LIN {X -0.012,Y -226.198,Z 1158.241,A 0.000,B 0.000,C 90.000,E1 43.380} C_DIS
LIN {X -0.070,Y -217.479,Z 1158.220,A 0.000,B 0.000,C 90.000,E1 39.564} C_DIS
LIN {X -0.002,Y -209.401,Z 1158.198,A 0.000,B 0.000,C 90.000,E1 35.644} C_DIS
LIN {X 0.014,Y -202.068,Z 1158.176,A 0.000,B 0.000,C 90.000,E1 31.671} C_DIS
LIN {X 0.064,Y -196.716,Z 1158.158,A 0.000,B 0.000,C 90.000,E1 28.437} C_DIS
LIN {X -0.032,Y -190.859,Z 1158.135,A 0.000,B 0.000,C 90.000,E1 24.387} C_DIS
LIN {X -0.001,Y -185.887,Z 1158.112,A 0.000,B 0.000,C 90.000,E1 20.248} C_DIS
LIN {X -0.022,Y -181.921,Z 1158.089,A 0.000,B 0.000,C 90.000,E1 16.079} C_DIS
LIN {X -0.067,Y -178.946,Z 1158.066,A 0.000,B 0.000,C 90.000,E1 11.883} C_DIS
LIN {X 0.040,Y -176.545,Z 1158.033,A 0.000,B 0.000,C 90.000,E1 5.910} C_DIS
LIN {X -0.034,Y -177.523,Z 1157.969,A 0.000,B 0.000,C 90.000,E1 354.432} C_DIS
LIN {X -0.032,Y -180.412,Z 1157.941,A 0.000,B 0.000,C 90.000,E1 349.342} C_DIS
LIN {X 0.053,Y -183.846,Z 1157.917,A 0.000,B 0.000,C 90.000,E1 345.102} C_DIS
LIN {X 0.088,Y -188.207,Z 1157.894,A 0.000,B 0.000,C 90.000,E1 340.913} C_DIS
LIN {X 0.033,Y -193.296,Z 1157.871,A 0.000,B 0.000,C 90.000,E1 336.794} C_DIS
LIN {X -0.094,Y -199.221,Z 1157.848,A 0.000,B 0.000,C 90.000,E1 332.743} C_DIS
LIN {X 0.072,Y -205.805,Z 1157.826,A 0.000,B 0.000,C 90.000,E1 328.663} C_DIS
LIN {X 0.075,Y -213.259,Z 1157.804,A 0.000,B 0.000,C 90.000,E1 324.689} C_DIS
LIN {X -0.021,Y -220.064,Z 1157.786,A 0.000,B 0.000,C 90.000,E1 321.582} C_DIS
LIN {X 0.021,Y -227.922,Z 1157.769,A 0.000,B 0.000,C 90.000,E1 318.485} C_DIS
LIN {X 0.025,Y -237.826,Z 1157.750,A 0.000,B 0.000,C 90.000,E1 315.081} C_DIS
LIN {X -0.014,Y -247.747,Z 1157.734,A 0.000,B 0.000,C 90.000,E1 312.123} C_DIS
LIN {X 0.041,Y -257.436,Z 1157.720,A 0.000,B 0.000,C 90.000,E1 309.564} C_DIS
LIN {X -0.005,Y -267.881,Z 1157.706,A 0.000,B 0.000,C 90.000,E1 307.076} C_DIS
LIN {X 0.126,Y -282.892,Z 1157.689,A 0.000,B 0.000,C 90.000,E1 303.913} C_DIS
LIN {X 0.086,Y -299.824,Z 1157.672,A 0.000,B 0.000,C 90.000,E1 300.875} C_DIS
LIN {X 0.078,Y -312.165,Z 1157.661,A 0.000,B 0.000,C 90.000,E1 298.899} C_DIS
LIN {X -0.128,Y -325.531,Z 1157.650,A 0.000,B 0.000,C 90.000,E1 297.001} C_DIS
LIN {X 0.004,Y -337.614,Z 1157.641,A 0.000,B 0.000,C 90.000,E1 295.412} C_DIS
LIN {X 0.021,Y -353.190,Z 1157.631,A 0.000,B 0.000,C 90.000,E1 293.567} C_DIS
LIN {X -0.118,Y -368.772,Z 1157.622,A 0.000,B 0.000,C 90.000,E1 291.972} C_DIS
LIN {X 0.035,Y -387.878,Z 1157.612,A 0.000,B 0.000,C 90.000,E1 290.174} C_DIS
LIN {X -0.171,Y -398.718,Z 1157.607,A 0.000,B 0.000,C 90.000,E1 289.214} C_DIS
LIN {X 0.062,Y -409.265,Z 1157.601,A 0.000,B 0.000,C 90.000,E1 288.181} C_DIS
LIN {X -0.151,Y -416.945,Z 1157.597,A 0.000,B 0.000,C 90.000,E1 287.457} C_DIS
LIN {X 0.059,Y -426.961,Z 1157.591,A 0.000,B 0.000,C 90.000,E1 286.386} C_DIS
LIN {X -0.111,Y -434.256,Z 1157.587,A 0.000,B 0.000,C 90.000,E1 285.607} C_DIS
LIN {X 0.144,Y -440.949,Z 1157.582,A 0.000,B 0.000,C 90.000,E1 284.773} C_DIS
LIN {X -0.071,Y -446.923,Z 1157.578,A 0.000,B 0.000,C 90.000,E1 284.008} C_DIS
LIN {X -0.137,Y -452.227,Z 1157.573,A 0.000,B 0.000,C 90.000,E1 283.231} C_DIS
LIN {X 0.186,Y -456.836,Z 1157.569,A 0.000,B 0.000,C 90.000,E1 282.411} C_DIS
LIN {X 0.008,Y -460.800,Z 1157.565,A 0.000,B 0.000,C 90.000,E1 281.658} C_DIS
LIN {X -0.036,Y -464.268,Z 1157.561,A 0.000,B 0.000,C 90.000,E1 280.894} C_DIS
LIN {X -0.142,Y -467.259,Z 1157.556,A 0.000,B 0.000,C 90.000,E1 280.141} C_DIS
LIN {X 0.005,Y -468.995,Z 1157.553,A 0.000,B 0.000,C 90.000,E1 279.613} C_DIS
LIN {X 0.087,Y -470.532,Z 1157.551,A 0.000,B 0.000,C 90.000,E1 279.095} C_DIS
LIN {X -0.214,Y -471.856,Z 1157.548,A 0.000,B 0.000,C 90.000,E1 278.624} C_DIS
LIN {X -0.111,Y -472.903,Z 1157.545,A 0.000,B 0.000,C 90.000,E1 278.106} C_DIS
LIN {X 0.001,Y -473.652,Z 1157.542,A 0.000,B 0.000,C 90.000,E1 277.587} C_DIS
LIN {X 0.122,Y -474.004,Z 1157.539,A 0.000,B 0.000,C 90.000,E1 277.068} C_DIS
LIN {X -0.222,Y -474.027,Z 1157.536,A 0.000,B 0.000,C 90.000,E1 276.606} C_DIS
LIN {X -0.095,Y -473.593,Z 1157.534,A 0.000,B 0.000,C 90.000,E1 276.087} C_DIS
LIN {X 0.033,Y -472.728,Z 1157.531,A 0.000,B 0.000,C 90.000,E1 275.568} C_DIS
LIN {X 0.156,Y -471.403,Z 1157.528,A 0.000,B 0.000,C 90.000,E1 275.049} C_DIS
LIN {X -0.196,Y -469.630,Z 1157.525,A 0.000,B 0.000,C 90.000,E1 274.588} C_DIS
LIN {X -0.123,Y -467.288,Z 1157.523,A 0.000,B 0.000,C 90.000,E1 274.073} C_DIS
LIN {X -0.032,Y -464.287,Z 1157.520,A 0.000,B 0.000,C 90.000,E1 273.555} C_DIS
LIN {X 0.039,Y -460.432,Z 1157.517,A 0.000,B 0.000,C 90.000,E1 273.037} C_DIS
LIN {X -0.177,Y -458.255,Z 1157.516,A 0.000,B 0.000,C 90.000,E1 272.808} C_DIS
LIN {X -0.080,Y -452.850,Z 1157.513,A 0.000,B 0.000,C 90.000,E1 272.293} C_DIS
LIN {X -0.220,Y -449.791,Z 1157.511,A 0.000,B 0.000,C 90.000,E1 272.064} C_DIS
LIN {X -0.132,Y -446.731,Z 1157.510,A 0.000,B 0.000,C 90.000,E1 271.835} C_DIS
LIN {X -0.085,Y -440.020,Z 1157.508,A 0.000,B 0.000,C 90.000,E1 271.432} C_DIS
LIN {X 0.061,Y -433.083,Z 1157.506,A 0.000,B 0.000,C 90.000,E1 271.088} C_DIS
LIN {X 0.186,Y -426.162,Z 1157.505,A 0.000,B 0.000,C 90.000,E1 270.802} C_DIS
LIN {X 0.201,Y -419.177,Z 1157.503,A 0.000,B 0.000,C 90.000,E1 270.573} C_DIS
LIN {X 0.062,Y -411.911,Z 1157.502,A 0.000,B 0.000,C 90.000,E1 270.401} C_DIS
LIN {X -0.006,Y -397.712,Z 1157.501,A 0.000,B 0.000,C 90.000,E1 270.115} C_DIS
LIN {X -0.055,Y -390.487,Z 1157.500,A 0.000,B 0.000,C 90.000,E1 270.000} C_DIS
LIN {X 0.012,Y -380.869,Z 1157.499,A 0.000,B 0.000,C 90.000,E1 269.885} C_DIS
LIN {X 0.159,Y -372.626,Z 1157.499,A 0.000,B 0.000,C 90.000,E1 269.828} C_DIS
LIN {X 0.060,Y -181.530,Z 1157.499,A 0.000,B 0.000,C 90.000,E1 269.828} C_DIS
LIN {X 0.006,Y -180.903,Z 1157.474,A 0.000,B 0.000,C 90.000,E1 265.298} C_DIS
LIN {X -0.045,Y -180.244,Z 1157.464,A 0.000,B 0.000,C 90.000,E1 263.628} C_DIS
LIN {X -0.026,Y -178.732,Z 1157.441,A 0.000,B 0.000,C 90.000,E1 259.398} C_DIS
LIN {X 0.042,Y -175.780,Z 1157.413,A 0.000,B 0.000,C 90.000,E1 254.283} C_DIS
LIN {X 0.029,Y -171.963,Z 1157.384,A 0.000,B 0.000,C 90.000,E1 249.156} C_DIS
LIN {X 0.067,Y -171.360,Z 1157.380,A 0.000,B 0.000,C 90.000,E1 248.284} C_DIS
LIN {X 0.044,Y -167.610,Z 1157.355,A 0.000,B 0.000,C 90.000,E1 243.973} C_DIS
LIN {X 0.056,Y -166.255,Z 1157.346,A 0.000,B 0.000,C 90.000,E1 242.231} C_DIS
LIN {X 0.044,Y -163.011,Z 1157.326,A 0.000,B 0.000,C 90.000,E1 238.742} C_DIS
LIN {X -0.044,Y -160.933,Z 1157.312,A 0.000,B 0.000,C 90.000,E1 236.135} C_DIS
LIN {X 0.067,Y -157.694,Z 1157.292,A 0.000,B 0.000,C 90.000,E1 232.557} C_DIS
LIN {X 0.005,Y -155.733,Z 1157.277,A 0.000,B 0.000,C 90.000,E1 229.908} C_DIS
LIN {X 0.058,Y -151.991,Z 1157.252,A 0.000,B 0.000,C 90.000,E1 225.405} C_DIS
LIN {X 0.074,Y -150.236,Z 1157.237,A 0.000,B 0.000,C 90.000,E1 222.690} C_DIS
LIN {X -0.003,Y -146.996,Z 1157.212,A 0.000,B 0.000,C 90.000,E1 218.177} C_DIS
LIN {X -0.013,Y -145.581,Z 1157.197,A 0.000,B 0.000,C 90.000,E1 215.438} C_DIS
LIN {X -0.019,Y -142.970,Z 1157.171,A 0.000,B 0.000,C 90.000,E1 210.846} C_DIS
LIN {X 0.035,Y -141.597,Z 1157.151,A 0.000,B 0.000,C 90.000,E1 207.129} C_DIS
LIN {X -0.050,Y -139.421,Z 1157.115,A 0.000,B 0.000,C 90.000,E1 200.663} C_DIS
LIN {X 0.001,Y -139.149,Z 1157.104,A 0.000,B 0.000,C 90.000,E1 198.779} C_DIS
LIN {X 0.023,Y -138.345,Z 1157.058,A 0.000,B 0.000,C 90.000,E1 190.366} C_DIS
LIN {X 0.009,Y -139.487,Z 1157.006,A 0.000,B 0.000,C 90.000,E1 181.031} C_DIS
LIN {X -0.051,Y -141.088,Z 1156.975,A 0.000,B 0.000,C 90.000,E1 175.469} C_DIS
LIN {X 0.044,Y -142.466,Z 1156.959,A 0.000,B 0.000,C 90.000,E1 172.648} C_DIS
LIN {X -0.008,Y -144.710,Z 1156.934,A 0.000,B 0.000,C 90.000,E1 168.049} C_DIS
LIN {X -0.057,Y -147.309,Z 1156.913,A 0.000,B 0.000,C 90.000,E1 164.393} C_DIS
LIN {X -0.042,Y -150.630,Z 1156.888,A 0.000,B 0.000,C 90.000,E1 159.826} C_DIS
LIN {X 0.035,Y -154.105,Z 1156.868,A 0.000,B 0.000,C 90.000,E1 156.177} C_DIS
LIN {X -0.041,Y -157.529,Z 1156.848,A 0.000,B 0.000,C 90.000,E1 152.615} C_DIS
LIN {X -0.098,Y -161.765,Z 1156.828,A 0.000,B 0.000,C 90.000,E1 149.076} C_DIS
LIN {X 0.008,Y -165.957,Z 1156.808,A 0.000,B 0.000,C 90.000,E1 145.515} C_DIS
LIN {X 0.005,Y -170.949,Z 1156.789,A 0.000,B 0.000,C 90.000,E1 142.029} C_DIS
LIN {X 0.057,Y -175.818,Z 1156.770,A 0.000,B 0.000,C 90.000,E1 138.566} C_DIS
LIN {X 0.052,Y -181.425,Z 1156.751,A 0.000,B 0.000,C 90.000,E1 135.162} C_DIS
LIN {X -0.074,Y -186.929,Z 1156.732,A 0.000,B 0.000,C 90.000,E1 131.838} C_DIS
LIN {X -0.001,Y -191.508,Z 1156.719,A 0.000,B 0.000,C 90.000,E1 129.322} C_DIS
LIN {X 0.083,Y -197.372,Z 1156.700,A 0.000,B 0.000,C 90.000,E1 126.011} C_DIS
LIN {X -0.067,Y -201.055,Z 1156.690,A 0.000,B 0.000,C 90.000,E1 124.199} C_DIS
LIN {X -0.152,Y -310.153,Z 1156.690,A 0.000,B 0.000,C 90.000,E1 124.199} C_DIS
LIN {X 0.183,Y -311.552,Z 1156.690,A 0.000,B 0.000,C 90.000,E1 124.119} C_DIS
LIN {X 0.058,Y -317.426,Z 1156.688,A 0.000,B 0.000,C 90.000,E1 123.865} C_DIS
LIN {X 0.109,Y -320.337,Z 1156.687,A 0.000,B 0.000,C 90.000,E1 123.579} C_DIS
LIN {X -0.149,Y -323.990,Z 1156.684,A 0.000,B 0.000,C 90.000,E1 123.086} C_DIS
LIN {X -0.066,Y -325.496,Z 1156.682,A 0.000,B 0.000,C 90.000,E1 122.752} C_DIS
LIN {X 0.007,Y -338.778,Z 1156.663,A 0.000,B 0.000,C 90.000,E1 119.283} C_DIS
LIN {X 0.175,Y -351.113,Z 1156.647,A 0.000,B 0.000,C 90.000,E1 116.488} C_DIS
LIN {X -0.101,Y -364.946,Z 1156.632,A 0.000,B 0.000,C 90.000,E1 113.823} C_DIS
LIN {X -0.071,Y -378.591,Z 1156.619,A 0.000,B 0.000,C 90.000,E1 111.461} C_DIS
LIN {X 0.029,Y -393.609,Z 1156.606,A 0.000,B 0.000,C 90.000,E1 109.141} C_DIS
LIN {X -0.129,Y -410.105,Z 1156.594,A 0.000,B 0.000,C 90.000,E1 106.913} C_DIS
LIN {X -0.116,Y -428.196,Z 1156.582,A 0.000,B 0.000,C 90.000,E1 104.717} C_DIS
LIN {X -0.033,Y -447.819,Z 1156.570,A 0.000,B 0.000,C 90.000,E1 102.591} C_DIS
LIN {X -0.186,Y -468.130,Z 1156.559,A 0.000,B 0.000,C 90.000,E1 100.658} C_DIS
LIN {X -0.149,Y -470.460,Z 1156.558,A 0.000,B 0.000,C 90.000,E1 100.423} C_DIS
LIN {X -0.198,Y -472.222,Z 1156.557,A 0.000,B 0.000,C 90.000,E1 100.197} C_DIS
LIN {X 0.125,Y -473.687,Z 1156.555,A 0.000,B 0.000,C 90.000,E1 99.905} C_DIS
LIN {X -0.019,Y -474.781,Z 1156.554,A 0.000,B 0.000,C 90.000,E1 99.670} C_DIS
LIN {X 0.100,Y -476.072,Z 1156.551,A 0.000,B 0.000,C 90.000,E1 99.151} C_DIS
LIN {X -0.170,Y -476.347,Z 1156.548,A 0.000,B 0.000,C 90.000,E1 98.681} C_DIS
LIN {X -0.036,Y -475.656,Z 1156.545,A 0.000,B 0.000,C 90.000,E1 98.163} C_DIS
LIN {X 0.103,Y -473.887,Z 1156.542,A 0.000,B 0.000,C 90.000,E1 97.644} C_DIS
LIN {X -0.034,Y -472.497,Z 1156.541,A 0.000,B 0.000,C 90.000,E1 97.409} C_DIS
LIN {X -0.121,Y -458.092,Z 1156.530,A 0.000,B 0.000,C 90.000,E1 95.391} C_DIS
LIN {X -0.197,Y -440.527,Z 1156.516,A 0.000,B 0.000,C 90.000,E1 92.808} C_DIS
LIN {X -0.102,Y -421.208,Z 1156.498,A 0.000,B 0.000,C 90.000,E1 89.599} C_DIS
LIN {X -0.043,Y -407.980,Z 1156.484,A 0.000,B 0.000,C 90.000,E1 87.135} C_DIS
LIN {X -0.042,Y -399.041,Z 1156.475,A 0.000,B 0.000,C 90.000,E1 85.469} C_DIS
LIN {X -0.104,Y -387.141,Z 1156.462,A 0.000,B 0.000,C 90.000,E1 83.223} C_DIS
LIN {X 0.012,Y -376.725,Z 1156.451,A 0.000,B 0.000,C 90.000,E1 81.197} C_DIS
LIN {X -0.011,Y -369.072,Z 1156.443,A 0.000,B 0.000,C 90.000,E1 79.746} C_DIS
LIN {X -0.114,Y -359.652,Z 1156.433,A 0.000,B 0.000,C 90.000,E1 77.993} C_DIS
LIN {X 0.036,Y -349.922,Z 1156.423,A 0.000,B 0.000,C 90.000,E1 76.172} C_DIS
LIN {X 0.080,Y -338.506,Z 1156.411,A 0.000,B 0.000,C 90.000,E1 74.031} C_DIS
LIN {X -0.155,Y -325.756,Z 1156.398,A 0.000,B 0.000,C 90.000,E1 71.583} C_DIS
LIN {X 0.094,Y -309.091,Z 1156.378,A 0.000,B 0.000,C 90.000,E1 68.028} C_DIS
LIN {X -0.021,Y -296.381,Z 1156.362,A 0.000,B 0.000,C 90.000,E1 65.101} C_DIS
LIN {X 0.048,Y -285.517,Z 1156.347,A 0.000,B 0.000,C 90.000,E1 62.410} C_DIS
LIN {X 0.058,Y -273.894,Z 1156.330,A 0.000,B 0.000,C 90.000,E1 59.331} C_DIS
LIN {X -0.071,Y -262.789,Z 1156.312,A 0.000,B 0.000,C 90.000,E1 56.215} C_DIS
LIN {X -0.067,Y -252.300,Z 1156.294,A 0.000,B 0.000,C 90.000,E1 53.004} C_DIS
LIN {X -0.137,Y -241.444,Z 1156.274,A 0.000,B 0.000,C 90.000,E1 49.380} C_DIS
LIN {X -0.063,Y -231.621,Z 1156.254,A 0.000,B 0.000,C 90.000,E1 45.648} C_DIS
LIN {X 0.021,Y -222.447,Z 1156.232,A 0.000,B 0.000,C 90.000,E1 41.838} C_DIS
LIN {X 0.043,Y -213.963,Z 1156.211,A 0.000,B 0.000,C 90.000,E1 37.971} C_DIS
LIN {X 0.043,Y -206.132,Z 1156.189,A 0.000,B 0.000,C 90.000,E1 34.040} C_DIS
LIN {X 0.018,Y -199.049,Z 1156.167,A 0.000,B 0.000,C 90.000,E1 30.050} C_DIS
LIN {X -0.025,Y -193.970,Z 1156.149,A 0.000,B 0.000,C 90.000,E1 26.821} C_DIS
LIN {X -0.017,Y -188.451,Z 1156.126,A 0.000,B 0.000,C 90.000,E1 22.717} C_DIS
LIN {X 0.051,Y -183.900,Z 1156.103,A 0.000,B 0.000,C 90.000,E1 18.544} C_DIS
LIN {X 0.034,Y -180.276,Z 1156.080,A 0.000,B 0.000,C 90.000,E1 14.356} C_DIS
LIN {X 0.086,Y -177.397,Z 1156.052,A 0.000,B 0.000,C 90.000,E1 9.265} C_DIS
LIN {X -0.091,Y -176.849,Z 1155.974,A 0.000,B 0.000,C 90.000,E1 355.298} C_DIS
LIN {X 0.060,Y -179.512,Z 1155.945,A 0.000,B 0.000,C 90.000,E1 350.151} C_DIS
LIN {X 0.038,Y -182.713,Z 1155.922,A 0.000,B 0.000,C 90.000,E1 345.936} C_DIS
LIN {X -0.019,Y -186.895,Z 1155.899,A 0.000,B 0.000,C 90.000,E1 341.764} C_DIS
LIN {X -0.013,Y -191.841,Z 1155.876,A 0.000,B 0.000,C 90.000,E1 337.614} C_DIS
LIN {X -0.012,Y -197.599,Z 1155.853,A 0.000,B 0.000,C 90.000,E1 333.512} C_DIS
LIN {X 0.007,Y -204.049,Z 1155.830,A 0.000,B 0.000,C 90.000,E1 329.459} C_DIS
LIN {X -0.109,Y -209.831,Z 1155.813,A 0.000,B 0.000,C 90.000,E1 326.294} C_DIS
LIN {X -0.083,Y -216.251,Z 1155.795,A 0.000,B 0.000,C 90.000,E1 323.130} C_DIS
LIN {X 0.027,Y -223.621,Z 1155.778,A 0.000,B 0.000,C 90.000,E1 319.989} C_DIS
LIN {X 0.080,Y -233.108,Z 1155.759,A 0.000,B 0.000,C 90.000,E1 316.539} C_DIS
LIN {X -0.054,Y -241.256,Z 1155.744,A 0.000,B 0.000,C 90.000,E1 313.947} C_DIS
LIN {X 0.006,Y -251.657,Z 1155.728,A 0.000,B 0.000,C 90.000,E1 310.987} C_DIS
LIN {X 0.089,Y -264.728,Z 1155.710,A 0.000,B 0.000,C 90.000,E1 307.729} C_DIS
LIN {X -0.096,Y -279.475,Z 1155.692,A 0.000,B 0.000,C 90.000,E1 304.612} C_DIS
LIN {X -0.044,Y -290.274,Z 1155.681,A 0.000,B 0.000,C 90.000,E1 302.546} C_DIS
LIN {X -0.059,Y -305.955,Z 1155.666,A 0.000,B 0.000,C 90.000,E1 299.873} C_DIS
LIN {X 0.033,Y -323.364,Z 1155.651,A 0.000,B 0.000,C 90.000,E1 297.257} C_DIS
LIN {X 0.107,Y -335.281,Z 1155.643,A 0.000,B 0.000,C 90.000,E1 295.668} C_DIS
LIN {X 0.089,Y -353.434,Z 1155.631,A 0.000,B 0.000,C 90.000,E1 293.515} C_DIS
LIN {X 0.152,Y -368.961,Z 1155.622,A 0.000,B 0.000,C 90.000,E1 291.897} C_DIS
LIN {X 0.183,Y -388.092,Z 1155.612,A 0.000,B 0.000,C 90.000,E1 290.120} C_DIS
LIN {X 0.163,Y -398.860,Z 1155.606,A 0.000,B 0.000,C 90.000,E1 289.141} C_DIS
LIN {X -0.095,Y -409.384,Z 1155.601,A 0.000,B 0.000,C 90.000,E1 288.181} C_DIS
LIN {X 0.085,Y -417.061,Z 1155.597,A 0.000,B 0.000,C 90.000,E1 287.402} C_DIS
LIN {X 0.070,Y -424.674,Z 1155.592,A 0.000,B 0.000,C 90.000,E1 286.622} C_DIS
LIN {X -0.043,Y -432.003,Z 1155.588,A 0.000,B 0.000,C 90.000,E1 285.843} C_DIS
LIN {X 0.199,Y -438.958,Z 1155.583,A 0.000,B 0.000,C 90.000,E1 285.009} C_DIS
LIN {X -0.041,Y -445.174,Z 1155.579,A 0.000,B 0.000,C 90.000,E1 284.245} C_DIS
LIN {X -0.114,Y -450.726,Z 1155.575,A 0.000,B 0.000,C 90.000,E1 283.467} C_DIS
LIN {X 0.190,Y -455.538,Z 1155.570,A 0.000,B 0.000,C 90.000,E1 282.647} C_DIS
LIN {X 0.099,Y -459.733,Z 1155.566,A 0.000,B 0.000,C 90.000,E1 281.883} C_DIS
LIN {X -0.052,Y -463.341,Z 1155.562,A 0.000,B 0.000,C 90.000,E1 281.130} C_DIS
LIN {X 0.141,Y -467.454,Z 1155.556,A 0.000,B 0.000,C 90.000,E1 280.084} C_DIS
LIN {X -0.172,Y -469.209,Z 1155.553,A 0.000,B 0.000,C 90.000,E1 279.613} C_DIS
LIN {X -0.089,Y -470.744,Z 1155.550,A 0.000,B 0.000,C 90.000,E1 279.095} C_DIS
LIN {X 0.078,Y -472.048,Z 1155.548,A 0.000,B 0.000,C 90.000,E1 278.568} C_DIS
LIN {X 0.183,Y -473.120,Z 1155.545,A 0.000,B 0.000,C 90.000,E1 278.049} C_DIS
LIN {X -0.172,Y -473.867,Z 1155.542,A 0.000,B 0.000,C 90.000,E1 277.587} C_DIS
LIN {X -0.050,Y -474.233,Z 1155.539,A 0.000,B 0.000,C 90.000,E1 277.068} C_DIS
LIN {X 0.077,Y -474.276,Z 1155.536,A 0.000,B 0.000,C 90.000,E1 276.549} C_DIS
LIN {X 0.207,Y -473.818,Z 1155.534,A 0.000,B 0.000,C 90.000,E1 276.030} C_DIS
LIN {X -0.135,Y -472.955,Z 1155.531,A 0.000,B 0.000,C 90.000,E1 275.568} C_DIS
LIN {X -0.010,Y -471.642,Z 1155.528,A 0.000,B 0.000,C 90.000,E1 275.049} C_DIS
LIN {X 0.107,Y -469.881,Z 1155.525,A 0.000,B 0.000,C 90.000,E1 274.531} C_DIS
LIN {X 0.214,Y -467.528,Z 1155.522,A 0.000,B 0.000,C 90.000,E1 274.012} C_DIS
LIN {X -0.191,Y -464.527,Z 1155.520,A 0.000,B 0.000,C 90.000,E1 273.555} C_DIS
LIN {X -0.118,Y -460.778,Z 1155.517,A 0.000,B 0.000,C 90.000,E1 273.037} C_DIS
LIN {X 0.126,Y -458.538,Z 1155.515,A 0.000,B 0.000,C 90.000,E1 272.751} C_DIS
LIN {X 0.221,Y -453.210,Z 1155.513,A 0.000,B 0.000,C 90.000,E1 272.236} C_DIS
LIN {X 0.187,Y -447.086,Z 1155.510,A 0.000,B 0.000,C 90.000,E1 271.776} C_DIS
LIN {X -0.214,Y -440.407,Z 1155.508,A 0.000,B 0.000,C 90.000,E1 271.432} C_DIS
LIN {X -0.072,Y -433.471,Z 1155.506,A 0.000,B 0.000,C 90.000,E1 271.088} C_DIS
LIN {X 0.041,Y -426.544,Z 1155.505,A 0.000,B 0.000,C 90.000,E1 270.802} C_DIS
LIN {X 0.053,Y -419.452,Z 1155.503,A 0.000,B 0.000,C 90.000,E1 270.573} C_DIS
LIN {X -0.088,Y -412.254,Z 1155.502,A 0.000,B 0.000,C 90.000,E1 270.401} C_DIS
LIN {X -0.087,Y -401.510,Z 1155.501,A 0.000,B 0.000,C 90.000,E1 270.172} C_DIS
LIN {X -0.189,Y -390.657,Z 1155.500,A 0.000,B 0.000,C 90.000,E1 270.000} C_DIS
LIN {X -0.113,Y -380.411,Z 1155.499,A 0.000,B 0.000,C 90.000,E1 269.885} C_DIS
LIN {X 0.114,Y -374.906,Z 1155.499,A 0.000,B 0.000,C 90.000,E1 269.828} C_DIS
LIN {X 0.020,Y -181.527,Z 1155.499,A 0.000,B 0.000,C 90.000,E1 269.828} C_DIS
LIN {X -0.052,Y -180.903,Z 1155.474,A 0.000,B 0.000,C 90.000,E1 265.298} C_DIS
LIN {X 0.078,Y -180.237,Z 1155.464,A 0.000,B 0.000,C 90.000,E1 263.571} C_DIS
LIN {X -0.082,Y -178.721,Z 1155.441,A 0.000,B 0.000,C 90.000,E1 259.398} C_DIS
LIN {X -0.013,Y -175.770,Z 1155.413,A 0.000,B 0.000,C 90.000,E1 254.283} C_DIS
LIN {X 0.036,Y -171.953,Z 1155.384,A 0.000,B 0.000,C 90.000,E1 249.135} C_DIS
LIN {X 0.012,Y -171.343,Z 1155.379,A 0.000,B 0.000,C 90.000,E1 248.284} C_DIS
LIN {X -0.009,Y -167.596,Z 1155.355,A 0.000,B 0.000,C 90.000,E1 243.973} C_DIS
LIN {X 0.003,Y -166.236,Z 1155.346,A 0.000,B 0.000,C 90.000,E1 242.231} C_DIS
LIN {X -0.009,Y -162.995,Z 1155.326,A 0.000,B 0.000,C 90.000,E1 238.742} C_DIS
LIN {X 0.038,Y -160.914,Z 1155.312,A 0.000,B 0.000,C 90.000,E1 236.087} C_DIS
LIN {X 0.015,Y -157.678,Z 1155.292,A 0.000,B 0.000,C 90.000,E1 232.557} C_DIS
LIN {X -0.046,Y -155.717,Z 1155.277,A 0.000,B 0.000,C 90.000,E1 229.908} C_DIS
LIN {X 0.008,Y -151.977,Z 1155.252,A 0.000,B 0.000,C 90.000,E1 225.405} C_DIS
LIN {X 0.024,Y -150.221,Z 1155.237,A 0.000,B 0.000,C 90.000,E1 222.690} C_DIS
LIN {X -0.052,Y -146.984,Z 1155.212,A 0.000,B 0.000,C 90.000,E1 218.177} C_DIS
LIN {X 0.057,Y -145.571,Z 1155.197,A 0.000,B 0.000,C 90.000,E1 215.391} C_DIS
LIN {X 0.056,Y -142.961,Z 1155.171,A 0.000,B 0.000,C 90.000,E1 210.797} C_DIS
LIN {X -0.014,Y -141.587,Z 1155.151,A 0.000,B 0.000,C 90.000,E1 207.129} C_DIS
LIN {X 0.033,Y -139.418,Z 1155.115,A 0.000,B 0.000,C 90.000,E1 200.610} C_DIS
LIN {X -0.047,Y -139.144,Z 1155.104,A 0.000,B 0.000,C 90.000,E1 198.779} C_DIS
LIN {X -0.025,Y -138.347,Z 1155.057,A 0.000,B 0.000,C 90.000,E1 190.366} C_DIS
LIN {X -0.039,Y -139.490,Z 1155.006,A 0.000,B 0.000,C 90.000,E1 181.031} C_DIS
LIN {X 0.042,Y -141.097,Z 1154.975,A 0.000,B 0.000,C 90.000,E1 175.412} C_DIS
LIN {X -0.005,Y -142.475,Z 1154.959,A 0.000,B 0.000,C 90.000,E1 172.648} C_DIS
LIN {X -0.058,Y -144.722,Z 1154.933,A 0.000,B 0.000,C 90.000,E1 168.049} C_DIS
LIN {X 0.035,Y -147.324,Z 1154.913,A 0.000,B 0.000,C 90.000,E1 164.338} C_DIS
LIN {X -0.040,Y -150.646,Z 1154.888,A 0.000,B 0.000,C 90.000,E1 159.806} C_DIS
LIN {X -0.017,Y -154.124,Z 1154.868,A 0.000,B 0.000,C 90.000,E1 156.177} C_DIS
LIN {X -0.094,Y -157.550,Z 1154.848,A 0.000,B 0.000,C 90.000,E1 152.615} C_DIS
LIN {X 0.071,Y -161.790,Z 1154.828,A 0.000,B 0.000,C 90.000,E1 148.997} C_DIS
LIN {X -0.046,Y -165.981,Z 1154.808,A 0.000,B 0.000,C 90.000,E1 145.515} C_DIS
LIN {X -0.051,Y -170.978,Z 1154.789,A 0.000,B 0.000,C 90.000,E1 142.029} C_DIS
LIN {X 0.000,Y -175.847,Z 1154.770,A 0.000,B 0.000,C 90.000,E1 138.566} C_DIS
LIN {X -0.005,Y -181.452,Z 1154.751,A 0.000,B 0.000,C 90.000,E1 135.162} C_DIS
LIN {X -0.007,Y -186.961,Z 1154.732,A 0.000,B 0.000,C 90.000,E1 131.800} C_DIS
LIN {X -0.011,Y -190.076,Z 1154.723,A 0.000,B 0.000,C 90.000,E1 130.135} C_DIS
LIN {X -0.119,Y -195.849,Z 1154.705,A 0.000,B 0.000,C 90.000,E1 126.870} C_DIS
LIN {X -0.096,Y -201.068,Z 1154.690,A 0.000,B 0.000,C 90.000,E1 124.199} C_DIS
LIN {X -0.196,Y -309.917,Z 1154.690,A 0.000,B 0.000,C 90.000,E1 124.199} C_DIS
LIN {X 0.089,Y -311.928,Z 1154.690,A 0.000,B 0.000,C 90.000,E1 124.119} C_DIS
LIN {X -0.037,Y -317.532,Z 1154.688,A 0.000,B 0.000,C 90.000,E1 123.865} C_DIS
LIN {X 0.013,Y -320.411,Z 1154.687,A 0.000,B 0.000,C 90.000,E1 123.579} C_DIS
LIN {X 0.000,Y -324.065,Z 1154.684,A 0.000,B 0.000,C 90.000,E1 123.038} C_DIS
LIN {X -0.189,Y -325.557,Z 1154.682,A 0.000,B 0.000,C 90.000,E1 122.752} C_DIS
LIN {X -0.119,Y -338.844,Z 1154.663,A 0.000,B 0.000,C 90.000,E1 119.283} C_DIS
LIN {X 0.047,Y -351.191,Z 1154.647,A 0.000,B 0.000,C 90.000,E1 116.488} C_DIS
LIN {X 0.101,Y -365.034,Z 1154.632,A 0.000,B 0.000,C 90.000,E1 113.770} C_DIS
LIN {X 0.148,Y -378.692,Z 1154.619,A 0.000,B 0.000,C 90.000,E1 111.408} C_DIS
LIN {X -0.107,Y -393.722,Z 1154.606,A 0.000,B 0.000,C 90.000,E1 109.141} C_DIS
LIN {X 0.125,Y -410.230,Z 1154.594,A 0.000,B 0.000,C 90.000,E1 106.858} C_DIS
LIN {X 0.155,Y -428.335,Z 1154.582,A 0.000,B 0.000,C 90.000,E1 104.662} C_DIS
LIN {X -0.174,Y -447.969,Z 1154.570,A 0.000,B 0.000,C 90.000,E1 102.591} C_DIS
LIN {X 0.137,Y -468.284,Z 1154.559,A 0.000,B 0.000,C 90.000,E1 100.602} C_DIS
LIN {X 0.176,Y -470.563,Z 1154.558,A 0.000,B 0.000,C 90.000,E1 100.366} C_DIS
LIN {X 0.132,Y -472.282,Z 1154.556,A 0.000,B 0.000,C 90.000,E1 100.141} C_DIS
LIN {X -0.011,Y -473.714,Z 1154.555,A 0.000,B 0.000,C 90.000,E1 99.905} C_DIS
LIN {X -0.155,Y -474.780,Z 1154.554,A 0.000,B 0.000,C 90.000,E1 99.670} C_DIS
LIN {X -0.036,Y -476.027,Z 1154.551,A 0.000,B 0.000,C 90.000,E1 99.151} C_DIS
LIN {X 0.165,Y -476.265,Z 1154.548,A 0.000,B 0.000,C 90.000,E1 98.624} C_DIS
LIN {X -0.171,Y -475.533,Z 1154.545,A 0.000,B 0.000,C 90.000,E1 98.163} C_DIS
LIN {X -0.033,Y -473.717,Z 1154.542,A 0.000,B 0.000,C 90.000,E1 97.644} C_DIS
LIN {X -0.169,Y -472.296,Z 1154.541,A 0.000,B 0.000,C 90.000,E1 97.409} C_DIS
LIN {X 0.198,Y -457.877,Z 1154.530,A 0.000,B 0.000,C 90.000,E1 95.334} C_DIS
LIN {X 0.107,Y -440.329,Z 1154.515,A 0.000,B 0.000,C 90.000,E1 92.751} C_DIS
LIN {X 0.182,Y -421.025,Z 1154.498,A 0.000,B 0.000,C 90.000,E1 89.542} C_DIS
LIN {X -0.181,Y -407.815,Z 1154.484,A 0.000,B 0.000,C 90.000,E1 87.135} C_DIS
LIN {X -0.179,Y -398.858,Z 1154.475,A 0.000,B 0.000,C 90.000,E1 85.469} C_DIS
LIN {X 0.142,Y -386.950,Z 1154.462,A 0.000,B 0.000,C 90.000,E1 83.166} C_DIS
LIN {X -0.125,Y -376.533,Z 1154.451,A 0.000,B 0.000,C 90.000,E1 81.197} C_DIS
LIN {X -0.150,Y -368.865,Z 1154.443,A 0.000,B 0.000,C 90.000,E1 79.746} C_DIS
LIN {X 0.099,Y -359.436,Z 1154.433,A 0.000,B 0.000,C 90.000,E1 77.937} C_DIS
LIN {X -0.103,Y -349.677,Z 1154.423,A 0.000,B 0.000,C 90.000,E1 76.172} C_DIS
LIN {X -0.060,Y -338.262,Z 1154.411,A 0.000,B 0.000,C 90.000,E1 74.031} C_DIS
LIN {X 0.118,Y -325.503,Z 1154.397,A 0.000,B 0.000,C 90.000,E1 71.511} C_DIS
LIN {X -0.047,Y -308.859,Z 1154.378,A 0.000,B 0.000,C 90.000,E1 68.028} C_DIS
LIN {X 0.107,Y -296.144,Z 1154.361,A 0.000,B 0.000,C 90.000,E1 65.049} C_DIS
LIN {X -0.094,Y -285.282,Z 1154.347,A 0.000,B 0.000,C 90.000,E1 62.410} C_DIS
LIN {X -0.084,Y -273.648,Z 1154.329,A 0.000,B 0.000,C 90.000,E1 59.331} C_DIS
LIN {X 0.004,Y -262.539,Z 1154.312,A 0.000,B 0.000,C 90.000,E1 56.167} C_DIS
LIN {X -0.036,Y -250.900,Z 1154.292,A 0.000,B 0.000,C 90.000,E1 52.603} C_DIS
LIN {X 0.057,Y -241.198,Z 1154.274,A 0.000,B 0.000,C 90.000,E1 49.299} C_DIS
LIN {X 0.116,Y -231.373,Z 1154.253,A 0.000,B 0.000,C 90.000,E1 45.567} C_DIS
LIN {X -0.130,Y -222.185,Z 1154.232,A 0.000,B 0.000,C 90.000,E1 41.838} C_DIS
LIN {X 0.022,Y -213.668,Z 1154.211,A 0.000,B 0.000,C 90.000,E1 37.935} C_DIS
LIN {X 0.058,Y -205.816,Z 1154.189,A 0.000,B 0.000,C 90.000,E1 33.992} C_DIS
LIN {X 0.029,Y -198.701,Z 1154.167,A 0.000,B 0.000,C 90.000,E1 30.001} C_DIS
LIN {X -0.092,Y -192.450,Z 1154.144,A 0.000,B 0.000,C 90.000,E1 25.976} C_DIS
LIN {X -0.037,Y -187.128,Z 1154.121,A 0.000,B 0.000,C 90.000,E1 21.844} C_DIS
LIN {X -0.075,Y -182.776,Z 1154.098,A 0.000,B 0.000,C 90.000,E1 17.692} C_DIS
LIN {X -0.006,Y -179.347,Z 1154.075,A 0.000,B 0.000,C 90.000,E1 13.467} C_DIS
LIN {X -0.001,Y -176.388,Z 1154.042,A 0.000,B 0.000,C 90.000,E1 7.530} C_DIS
LIN {X -0.029,Y -177.248,Z 1153.964,A 0.000,B 0.000,C 90.000,E1 353.571} C_DIS
LIN {X 0.013,Y -180.341,Z 1153.936,A 0.000,B 0.000,C 90.000,E1 348.465} C_DIS
LIN {X -0.037,Y -183.889,Z 1153.912,A 0.000,B 0.000,C 90.000,E1 344.267} C_DIS
LIN {X 0.056,Y -188.402,Z 1153.889,A 0.000,B 0.000,C 90.000,E1 340.061} C_DIS
LIN {X 0.078,Y -193.668,Z 1153.866,A 0.000,B 0.000,C 90.000,E1 335.921} C_DIS
LIN {X 0.048,Y -199.705,Z 1153.844,A 0.000,B 0.000,C 90.000,E1 331.847} C_DIS
LIN {X -0.017,Y -206.493,Z 1153.821,A 0.000,B 0.000,C 90.000,E1 327.837} C_DIS
LIN {X 0.040,Y -212.643,Z 1153.804,A 0.000,B 0.000,C 90.000,E1 324.642} C_DIS
LIN {X -0.080,Y -219.568,Z 1153.786,A 0.000,B 0.000,C 90.000,E1 321.537} C_DIS
LIN {X 0.007,Y -226.449,Z 1153.771,A 0.000,B 0.000,C 90.000,E1 318.809} C_DIS
LIN {X -0.040,Y -236.302,Z 1153.752,A 0.000,B 0.000,C 90.000,E1 315.405} C_DIS
LIN {X -0.120,Y -246.169,Z 1153.736,A 0.000,B 0.000,C 90.000,E1 312.447} C_DIS
LIN {X 0.091,Y -257.261,Z 1153.719,A 0.000,B 0.000,C 90.000,E1 309.483} C_DIS
LIN {X 0.041,Y -267.826,Z 1153.706,A 0.000,B 0.000,C 90.000,E1 306.996} C_DIS
LIN {X 0.012,Y -283.001,Z 1153.688,A 0.000,B 0.000,C 90.000,E1 303.865} C_DIS
LIN {X 0.132,Y -300.028,Z 1153.671,A 0.000,B 0.000,C 90.000,E1 300.797} C_DIS
LIN {X 0.127,Y -312.427,Z 1153.660,A 0.000,B 0.000,C 90.000,E1 298.821} C_DIS
LIN {X -0.143,Y -328.182,Z 1153.648,A 0.000,B 0.000,C 90.000,E1 296.616} C_DIS
LIN {X 0.016,Y -343.053,Z 1153.637,A 0.000,B 0.000,C 90.000,E1 294.719} C_DIS
LIN {X -0.119,Y -355.963,Z 1153.629,A 0.000,B 0.000,C 90.000,E1 293.259} C_DIS
LIN {X -0.015,Y -369.096,Z 1153.622,A 0.000,B 0.000,C 90.000,E1 291.897} C_DIS
LIN {X 0.018,Y -388.220,Z 1153.612,A 0.000,B 0.000,C 90.000,E1 290.120} C_DIS
LIN {X -0.023,Y -399.019,Z 1153.606,A 0.000,B 0.000,C 90.000,E1 289.141} C_DIS
LIN {X 0.143,Y -409.512,Z 1153.601,A 0.000,B 0.000,C 90.000,E1 288.127} C_DIS
LIN {X -0.132,Y -417.273,Z 1153.597,A 0.000,B 0.000,C 90.000,E1 287.402} C_DIS
LIN {X 0.179,Y -427.386,Z 1153.591,A 0.000,B 0.000,C 90.000,E1 286.315} C_DIS
LIN {X -0.092,Y -434.638,Z 1153.586,A 0.000,B 0.000,C 90.000,E1 285.552} C_DIS
LIN {X 0.169,Y -441.352,Z 1153.582,A 0.000,B 0.000,C 90.000,E1 284.717} C_DIS
LIN {X 0.066,Y -447.341,Z 1153.578,A 0.000,B 0.000,C 90.000,E1 283.939} C_DIS
LIN {X -0.101,Y -452.621,Z 1153.573,A 0.000,B 0.000,C 90.000,E1 283.175} C_DIS
LIN {X 0.226,Y -457.261,Z 1153.569,A 0.000,B 0.000,C 90.000,E1 282.355} C_DIS
LIN {X 0.147,Y -461.247,Z 1153.564,A 0.000,B 0.000,C 90.000,E1 281.591} C_DIS
LIN {X -0.148,Y -465.736,Z 1153.559,A 0.000,B 0.000,C 90.000,E1 280.602} C_DIS
LIN {X -0.005,Y -467.688,Z 1153.556,A 0.000,B 0.000,C 90.000,E1 280.074} C_DIS
LIN {X 0.065,Y -469.443,Z 1153.553,A 0.000,B 0.000,C 90.000,E1 279.557} C_DIS
LIN {X 0.224,Y -470.980,Z 1153.550,A 0.000,B 0.000,C 90.000,E1 279.029} C_DIS
LIN {X -0.147,Y -472.314,Z 1153.547,A 0.000,B 0.000,C 90.000,E1 278.568} C_DIS
LIN {X -0.041,Y -473.371,Z 1153.545,A 0.000,B 0.000,C 90.000,E1 278.049} C_DIS
LIN {X 0.074,Y -474.089,Z 1153.542,A 0.000,B 0.000,C 90.000,E1 277.530} C_DIS
LIN {X 0.199,Y -474.493,Z 1153.539,A 0.000,B 0.000,C 90.000,E1 277.011} C_DIS
LIN {X -0.089,Y -474.480,Z 1153.536,A 0.000,B 0.000,C 90.000,E1 276.543} C_DIS
LIN {X -0.012,Y -474.058,Z 1153.533,A 0.000,B 0.000,C 90.000,E1 276.030} C_DIS
LIN {X 0.119,Y -473.181,Z 1153.531,A 0.000,B 0.000,C 90.000,E1 275.511} C_DIS
LIN {X -0.225,Y -471.879,Z 1153.528,A 0.000,B 0.000,C 90.000,E1 275.049} C_DIS
LIN {X -0.105,Y -470.107,Z 1153.525,A 0.000,B 0.000,C 90.000,E1 274.531} C_DIS
LIN {X 0.004,Y -467.775,Z 1153.522,A 0.000,B 0.000,C 90.000,E1 274.012} C_DIS
LIN {X 0.064,Y -464.809,Z 1153.520,A 0.000,B 0.000,C 90.000,E1 273.498} C_DIS
LIN {X 0.137,Y -461.045,Z 1153.517,A 0.000,B 0.000,C 90.000,E1 272.980} C_DIS
LIN {X -0.078,Y -458.794,Z 1153.515,A 0.000,B 0.000,C 90.000,E1 272.751} C_DIS
LIN {X 0.005,Y -453.469,Z 1153.512,A 0.000,B 0.000,C 90.000,E1 272.236} C_DIS
LIN {X -0.153,Y -450.333,Z 1153.511,A 0.000,B 0.000,C 90.000,E1 272.007} C_DIS
LIN {X 0.076,Y -443.824,Z 1153.509,A 0.000,B 0.000,C 90.000,E1 271.547} C_DIS
LIN {X -0.044,Y -436.945,Z 1153.507,A 0.000,B 0.000,C 90.000,E1 271.203} C_DIS
LIN {X -0.119,Y -429.969,Z 1153.505,A 0.000,B 0.000,C 90.000,E1 270.917} C_DIS
LIN {X 0.175,Y -422.883,Z 1153.504,A 0.000,B 0.000,C 90.000,E1 270.630} C_DIS
LIN {X -0.072,Y -415.729,Z 1153.502,A 0.000,B 0.000,C 90.000,E1 270.458} C_DIS
LIN {X -0.175,Y -405.067,Z 1153.501,A 0.000,B 0.000,C 90.000,E1 270.229} C_DIS
LIN {X 0.021,Y -394.228,Z 1153.500,A 0.000,B 0.000,C 90.000,E1 270.000} C_DIS
LIN {X 0.041,Y -385.617,Z 1153.499,A 0.000,B 0.000,C 90.000,E1 269.885} C_DIS
LIN {X -0.004,Y -373.609,Z 1153.499,A 0.000,B 0.000,C 90.000,E1 269.828} C_DIS
LIN {X -0.035,Y -181.523,Z 1153.499,A 0.000,B 0.000,C 90.000,E1 269.828} C_DIS
LIN {X 0.078,Y -180.902,Z 1153.474,A 0.000,B 0.000,C 90.000,E1 265.241} C_DIS
LIN {X 0.028,Y -180.229,Z 1153.464,A 0.000,B 0.000,C 90.000,E1 263.571} C_DIS
LIN {X -0.019,Y -179.042,Z 1153.446,A 0.000,B 0.000,C 90.000,E1 260.208} C_DIS
LIN {X 0.044,Y -178.711,Z 1153.441,A 0.000,B 0.000,C 90.000,E1 259.342} C_DIS
LIN {X -0.064,Y -175.760,Z 1153.413,A 0.000,B 0.000,C 90.000,E1 254.283} C_DIS
LIN {X -0.013,Y -171.943,Z 1153.384,A 0.000,B 0.000,C 90.000,E1 249.135} C_DIS
LIN {X -0.037,Y -171.328,Z 1153.379,A 0.000,B 0.000,C 90.000,E1 248.284} C_DIS
LIN {X 0.015,Y -167.584,Z 1153.355,A 0.000,B 0.000,C 90.000,E1 243.948} C_DIS
LIN {X -0.046,Y -166.220,Z 1153.346,A 0.000,B 0.000,C 90.000,E1 242.231} C_DIS
LIN {X -0.057,Y -162.982,Z 1153.326,A 0.000,B 0.000,C 90.000,E1 238.742} C_DIS
LIN {X -0.009,Y -160.897,Z 1153.312,A 0.000,B 0.000,C 90.000,E1 236.087} C_DIS
LIN {X -0.031,Y -157.664,Z 1153.292,A 0.000,B 0.000,C 90.000,E1 232.557} C_DIS
LIN {X -0.093,Y -155.702,Z 1153.277,A 0.000,B 0.000,C 90.000,E1 229.908} C_DIS
LIN {X -0.037,Y -151.966,Z 1153.252,A 0.000,B 0.000,C 90.000,E1 225.405} C_DIS
LIN {X -0.021,Y -150.208,Z 1153.237,A 0.000,B 0.000,C 90.000,E1 222.690} C_DIS
LIN {X -0.006,Y -146.975,Z 1153.212,A 0.000,B 0.000,C 90.000,E1 218.141} C_DIS
LIN {X 0.012,Y -145.561,Z 1153.197,A 0.000,B 0.000,C 90.000,E1 215.391} C_DIS
LIN {X 0.012,Y -142.953,Z 1153.171,A 0.000,B 0.000,C 90.000,E1 210.797} C_DIS
LIN {X -0.057,Y -141.579,Z 1153.151,A 0.000,B 0.000,C 90.000,E1 207.129} C_DIS
LIN {X -0.010,Y -139.415,Z 1153.115,A 0.000,B 0.000,C 90.000,E1 200.610} C_DIS
LIN {X 0.042,Y -139.140,Z 1153.104,A 0.000,B 0.000,C 90.000,E1 198.725} C_DIS
LIN {X 0.068,Y -138.348,Z 1153.057,A 0.000,B 0.000,C 90.000,E1 190.310} C_DIS
LIN {X 0.057,Y -139.492,Z 1153.005,A 0.000,B 0.000,C 90.000,E1 180.974} C_DIS
LIN {X -0.002,Y -141.104,Z 1152.974,A 0.000,B 0.000,C 90.000,E1 175.412} C_DIS
LIN {X -0.049,Y -142.483,Z 1152.959,A 0.000,B 0.000,C 90.000,E1 172.648} C_DIS
LIN {X 0.040,Y -144.733,Z 1152.933,A 0.000,B 0.000,C 90.000,E1 167.993} C_DIS
LIN {X -0.010,Y -147.337,Z 1152.913,A 0.000,B 0.000,C 90.000,E1 164.338} C_DIS
LIN {X 0.055,Y -150.661,Z 1152.888,A 0.000,B 0.000,C 90.000,E1 159.752} C_DIS
LIN {X -0.063,Y -154.139,Z 1152.868,A 0.000,B 0.000,C 90.000,E1 156.177} C_DIS
LIN {X -0.001,Y -157.568,Z 1152.848,A 0.000,B 0.000,C 90.000,E1 152.564} C_DIS
LIN {X 0.024,Y -161.811,Z 1152.828,A 0.000,B 0.000,C 90.000,E1 148.997} C_DIS
LIN {X 0.042,Y -166.003,Z 1152.808,A 0.000,B 0.000,C 90.000,E1 145.468} C_DIS
LIN {X 0.035,Y -171.001,Z 1152.789,A 0.000,B 0.000,C 90.000,E1 141.984} C_DIS
LIN {X -0.050,Y -175.872,Z 1152.770,A 0.000,B 0.000,C 90.000,E1 138.566} C_DIS
LIN {X -0.056,Y -181.476,Z 1152.751,A 0.000,B 0.000,C 90.000,E1 135.162} C_DIS
LIN {X 0.081,Y -186.990,Z 1152.732,A 0.000,B 0.000,C 90.000,E1 131.757} C_DIS
LIN {X 0.083,Y -190.106,Z 1152.723,A 0.000,B 0.000,C 90.000,E1 130.092} C_DIS
LIN {X 0.102,Y -195.878,Z 1152.705,A 0.000,B 0.000,C 90.000,E1 126.790} C_DIS
LIN {X 0.130,Y -201.094,Z 1152.690,A 0.000,B 0.000,C 90.000,E1 124.119} C_DIS
LIN {X 0.151,Y -309.939,Z 1152.690,A 0.000,B 0.000,C 90.000,E1 124.119} C_DIS
LIN {X 0.006,Y -311.957,Z 1152.690,A 0.000,B 0.000,C 90.000,E1 124.119} C_DIS
LIN {X 0.055,Y -317.561,Z 1152.688,A 0.000,B 0.000,C 90.000,E1 123.833} C_DIS
LIN {X -0.073,Y -320.443,Z 1152.687,A 0.000,B 0.000,C 90.000,E1 123.579} C_DIS
LIN {X -0.086,Y -324.096,Z 1152.683,A 0.000,B 0.000,C 90.000,E1 123.038} C_DIS
LIN {X -0.002,Y -325.589,Z 1152.682,A 0.000,B 0.000,C 90.000,E1 122.704} C_DIS
LIN {X -0.042,Y -338.884,Z 1152.662,A 0.000,B 0.000,C 90.000,E1 119.255} C_DIS
LIN {X -0.043,Y -351.238,Z 1152.647,A 0.000,B 0.000,C 90.000,E1 116.488} C_DIS
LIN {X 0.008,Y -365.091,Z 1152.632,A 0.000,B 0.000,C 90.000,E1 113.770} C_DIS
LIN {X 0.053,Y -378.756,Z 1152.619,A 0.000,B 0.000,C 90.000,E1 111.408} C_DIS
LIN {X 0.168,Y -393.794,Z 1152.606,A 0.000,B 0.000,C 90.000,E1 109.087} C_DIS
LIN {X 0.025,Y -410.313,Z 1152.594,A 0.000,B 0.000,C 90.000,E1 106.858} C_DIS
LIN {X 0.054,Y -428.428,Z 1152.582,A 0.000,B 0.000,C 90.000,E1 104.662} C_DIS
LIN {X 0.162,Y -448.068,Z 1152.570,A 0.000,B 0.000,C 90.000,E1 102.535} C_DIS
LIN {X 0.039,Y -468.388,Z 1152.559,A 0.000,B 0.000,C 90.000,E1 100.602} C_DIS
LIN {X 0.079,Y -470.627,Z 1152.558,A 0.000,B 0.000,C 90.000,E1 100.366} C_DIS
LIN {X 0.035,Y -472.318,Z 1152.556,A 0.000,B 0.000,C 90.000,E1 100.141} C_DIS
LIN {X -0.107,Y -473.727,Z 1152.555,A 0.000,B 0.000,C 90.000,E1 99.905} C_DIS
LIN {X 0.216,Y -474.774,Z 1152.554,A 0.000,B 0.000,C 90.000,E1 99.613} C_DIS
LIN {X -0.133,Y -475.989,Z 1152.551,A 0.000,B 0.000,C 90.000,E1 99.151} C_DIS
LIN {X 0.067,Y -476.199,Z 1152.548,A 0.000,B 0.000,C 90.000,E1 98.624} C_DIS
LIN {X 0.201,Y -475.439,Z 1152.545,A 0.000,B 0.000,C 90.000,E1 98.106} C_DIS
LIN {X -0.131,Y -473.589,Z 1152.542,A 0.000,B 0.000,C 90.000,E1 97.644} C_DIS
LIN {X 0.201,Y -472.145,Z 1152.541,A 0.000,B 0.000,C 90.000,E1 97.352} C_DIS
LIN {X -0.123,Y -455.879,Z 1152.528,A 0.000,B 0.000,C 90.000,E1 95.106} C_DIS
LIN {X 0.186,Y -438.508,Z 1152.514,A 0.000,B 0.000,C 90.000,E1 92.465} C_DIS
LIN {X 0.082,Y -420.870,Z 1152.498,A 0.000,B 0.000,C 90.000,E1 89.542} C_DIS
LIN {X 0.125,Y -407.675,Z 1152.484,A 0.000,B 0.000,C 90.000,E1 87.078} C_DIS
LIN {X 0.118,Y -398.699,Z 1152.475,A 0.000,B 0.000,C 90.000,E1 85.412} C_DIS
LIN {X 0.040,Y -386.786,Z 1152.462,A 0.000,B 0.000,C 90.000,E1 83.166} C_DIS
LIN {X 0.144,Y -376.383,Z 1152.451,A 0.000,B 0.000,C 90.000,E1 81.141} C_DIS
LIN {X 0.100,Y -367.128,Z 1152.441,A 0.000,B 0.000,C 90.000,E1 79.398} C_DIS
LIN {X -0.042,Y -357.643,Z 1152.431,A 0.000,B 0.000,C 90.000,E1 77.645} C_DIS
LIN {X 0.065,Y -347.845,Z 1152.421,A 0.000,B 0.000,C 90.000,E1 75.825} C_DIS
LIN {X 0.061,Y -336.420,Z 1152.409,A 0.000,B 0.000,C 90.000,E1 73.685} C_DIS
LIN {X -0.130,Y -323.701,Z 1152.396,A 0.000,B 0.000,C 90.000,E1 71.221} C_DIS
LIN {X 0.042,Y -307.219,Z 1152.376,A 0.000,B 0.000,C 90.000,E1 67.667} C_DIS
LIN {X 0.000,Y -294.561,Z 1152.359,A 0.000,B 0.000,C 90.000,E1 64.717} C_DIS
LIN {X 0.023,Y -283.744,Z 1152.345,A 0.000,B 0.000,C 90.000,E1 62.025} C_DIS
LIN {X 0.038,Y -273.425,Z 1152.329,A 0.000,B 0.000,C 90.000,E1 59.282} C_DIS
LIN {X -0.054,Y -261.094,Z 1152.310,A 0.000,B 0.000,C 90.000,E1 55.801} C_DIS
LIN {X 0.047,Y -250.653,Z 1152.292,A 0.000,B 0.000,C 90.000,E1 52.557} C_DIS
LIN {X -0.062,Y -240.968,Z 1152.274,A 0.000,B 0.000,C 90.000,E1 49.299} C_DIS
LIN {X -0.005,Y -231.140,Z 1152.253,A 0.000,B 0.000,C 90.000,E1 45.567} C_DIS
LIN {X 0.061,Y -221.938,Z 1152.232,A 0.000,B 0.000,C 90.000,E1 41.757} C_DIS
LIN {X 0.064,Y -213.389,Z 1152.211,A 0.000,B 0.000,C 90.000,E1 37.890} C_DIS
LIN {X -0.072,Y -205.514,Z 1152.189,A 0.000,B 0.000,C 90.000,E1 33.992} C_DIS
LIN {X -0.106,Y -198.365,Z 1152.167,A 0.000,B 0.000,C 90.000,E1 30.001} C_DIS
LIN {X 0.025,Y -192.111,Z 1152.144,A 0.000,B 0.000,C 90.000,E1 25.899} C_DIS
LIN {X 0.059,Y -186.818,Z 1152.121,A 0.000,B 0.000,C 90.000,E1 21.770} C_DIS
LIN {X -0.054,Y -182.453,Z 1152.098,A 0.000,B 0.000,C 90.000,E1 17.638} C_DIS
LIN {X 0.009,Y -179.025,Z 1152.074,A 0.000,B 0.000,C 90.000,E1 13.411} C_DIS
LIN {X 0.026,Y -176.051,Z 1152.042,A 0.000,B 0.000,C 90.000,E1 7.466} C_DIS
LIN {X -0.043,Y -176.918,Z 1151.964,A 0.000,B 0.000,C 90.000,E1 353.571} C_DIS
LIN {X -0.013,Y -180.005,Z 1151.936,A 0.000,B 0.000,C 90.000,E1 348.465} C_DIS
LIN {X 0.102,Y -183.548,Z 1151.912,A 0.000,B 0.000,C 90.000,E1 344.212} C_DIS
LIN {X 0.006,Y -188.026,Z 1151.889,A 0.000,B 0.000,C 90.000,E1 340.061} C_DIS
LIN {X 0.015,Y -193.298,Z 1151.866,A 0.000,B 0.000,C 90.000,E1 335.921} C_DIS
LIN {X -0.030,Y -199.316,Z 1151.844,A 0.000,B 0.000,C 90.000,E1 331.847} C_DIS
LIN {X -0.021,Y -204.711,Z 1151.826,A 0.000,B 0.000,C 90.000,E1 328.614} C_DIS
LIN {X 0.104,Y -210.740,Z 1151.808,A 0.000,B 0.000,C 90.000,E1 325.388} C_DIS
LIN {X -0.016,Y -217.482,Z 1151.790,A 0.000,B 0.000,C 90.000,E1 322.271} C_DIS
LIN {X -0.049,Y -225.180,Z 1151.773,A 0.000,B 0.000,C 90.000,E1 319.175} C_DIS
LIN {X 0.040,Y -234.981,Z 1151.754,A 0.000,B 0.000,C 90.000,E1 315.729} C_DIS
LIN {X -0.070,Y -244.744,Z 1151.738,A 0.000,B 0.000,C 90.000,E1 312.771} C_DIS
LIN {X -0.087,Y -255.709,Z 1151.721,A 0.000,B 0.000,C 90.000,E1 309.850} C_DIS
LIN {X 0.028,Y -266.181,Z 1151.707,A 0.000,B 0.000,C 90.000,E1 307.317} C_DIS
LIN {X -0.106,Y -281.258,Z 1151.690,A 0.000,B 0.000,C 90.000,E1 304.199} C_DIS
LIN {X -0.018,Y -292.326,Z 1151.678,A 0.000,B 0.000,C 90.000,E1 302.133} C_DIS
LIN {X -0.012,Y -306.187,Z 1151.666,A 0.000,B 0.000,C 90.000,E1 299.795} C_DIS
LIN {X -0.065,Y -323.646,Z 1151.651,A 0.000,B 0.000,C 90.000,E1 297.206} C_DIS
LIN {X 0.154,Y -335.579,Z 1151.642,A 0.000,B 0.000,C 90.000,E1 295.591} C_DIS
LIN {X -0.124,Y -353.496,Z 1151.630,A 0.000,B 0.000,C 90.000,E1 293.515} C_DIS
LIN {X -0.134,Y -364.190,Z 1151.624,A 0.000,B 0.000,C 90.000,E1 292.386} C_DIS
LIN {X -0.089,Y -388.830,Z 1151.611,A 0.000,B 0.000,C 90.000,E1 290.066} C_DIS
LIN {X -0.105,Y -399.618,Z 1151.606,A 0.000,B 0.000,C 90.000,E1 289.087} C_DIS
LIN {X 0.195,Y -410.075,Z 1151.600,A 0.000,B 0.000,C 90.000,E1 288.055} C_DIS
LIN {X -0.052,Y -417.806,Z 1151.596,A 0.000,B 0.000,C 90.000,E1 287.330} C_DIS
LIN {X 0.141,Y -427.895,Z 1151.590,A 0.000,B 0.000,C 90.000,E1 286.260} C_DIS
LIN {X 0.156,Y -437.446,Z 1151.584,A 0.000,B 0.000,C 90.000,E1 285.190} C_DIS
LIN {X 0.022,Y -443.923,Z 1151.580,A 0.000,B 0.000,C 90.000,E1 284.411} C_DIS
LIN {X -0.178,Y -449.629,Z 1151.576,A 0.000,B 0.000,C 90.000,E1 283.647} C_DIS
LIN {X 0.121,Y -454.652,Z 1151.571,A 0.000,B 0.000,C 90.000,E1 282.827} C_DIS
LIN {X 0.019,Y -459.024,Z 1151.567,A 0.000,B 0.000,C 90.000,E1 282.063} C_DIS
LIN {X -0.042,Y -462.810,Z 1151.563,A 0.000,B 0.000,C 90.000,E1 281.299} C_DIS
LIN {X -0.164,Y -466.100,Z 1151.558,A 0.000,B 0.000,C 90.000,E1 280.546} C_DIS
LIN {X -0.019,Y -468.046,Z 1151.556,A 0.000,B 0.000,C 90.000,E1 280.018} C_DIS
LIN {X 0.054,Y -469.804,Z 1151.553,A 0.000,B 0.000,C 90.000,E1 279.500} C_DIS
LIN {X 0.215,Y -471.345,Z 1151.550,A 0.000,B 0.000,C 90.000,E1 278.973} C_DIS
LIN {X -0.153,Y -472.627,Z 1151.547,A 0.000,B 0.000,C 90.000,E1 278.511} C_DIS
LIN {X -0.044,Y -473.659,Z 1151.544,A 0.000,B 0.000,C 90.000,E1 277.992} C_DIS
LIN {X 0.075,Y -474.341,Z 1151.542,A 0.000,B 0.000,C 90.000,E1 277.473} C_DIS
LIN {X 0.259,Y -474.707,Z 1151.539,A 0.000,B 0.000,C 90.000,E1 276.947} C_DIS
LIN {X -0.086,Y -474.672,Z 1151.536,A 0.000,B 0.000,C 90.000,E1 276.486} C_DIS
LIN {X 0.043,Y -474.228,Z 1151.533,A 0.000,B 0.000,C 90.000,E1 275.967} C_DIS
LIN {X 0.126,Y -473.340,Z 1151.530,A 0.000,B 0.000,C 90.000,E1 275.454} C_DIS
LIN {X -0.217,Y -472.025,Z 1151.528,A 0.000,B 0.000,C 90.000,E1 274.992} C_DIS
LIN {X -0.096,Y -470.202,Z 1151.525,A 0.000,B 0.000,C 90.000,E1 274.473} C_DIS
LIN {X 0.014,Y -467.862,Z 1151.522,A 0.000,B 0.000,C 90.000,E1 273.955} C_DIS
LIN {X 0.076,Y -464.883,Z 1151.519,A 0.000,B 0.000,C 90.000,E1 273.440} C_DIS
LIN {X 0.149,Y -461.072,Z 1151.516,A 0.000,B 0.000,C 90.000,E1 272.922} C_DIS
LIN {X 0.178,Y -456.190,Z 1151.514,A 0.000,B 0.000,C 90.000,E1 272.407} C_DIS
LIN {X 0.022,Y -453.374,Z 1151.512,A 0.000,B 0.000,C 90.000,E1 272.178} C_DIS
LIN {X -0.132,Y -450.220,Z 1151.511,A 0.000,B 0.000,C 90.000,E1 271.949} C_DIS
LIN {X 0.000,Y -447.136,Z 1151.510,A 0.000,B 0.000,C 90.000,E1 271.718} C_DIS
LIN {X 0.086,Y -440.362,Z 1151.507,A 0.000,B 0.000,C 90.000,E1 271.318} C_DIS
LIN {X -0.184,Y -433.442,Z 1151.506,A 0.000,B 0.000,C 90.000,E1 271.031} C_DIS
LIN {X -0.057,Y -426.407,Z 1151.504,A 0.000,B 0.000,C 90.000,E1 270.745} C_DIS
LIN {X -0.024,Y -419.150,Z 1151.503,A 0.000,B 0.000,C 90.000,E1 270.516} C_DIS
LIN {X 0.088,Y -408.209,Z 1151.501,A 0.000,B 0.000,C 90.000,E1 270.229} C_DIS
LIN {X -0.153,Y -397.781,Z 1151.500,A 0.000,B 0.000,C 90.000,E1 270.057} C_DIS
LIN {X -0.161,Y -390.173,Z 1151.500,A 0.000,B 0.000,C 90.000,E1 269.943} C_DIS
LIN {X 0.120,Y -382.030,Z 1151.499,A 0.000,B 0.000,C 90.000,E1 269.828} C_DIS
LIN {X -0.078,Y -374.328,Z 1151.499,A 0.000,B 0.000,C 90.000,E1 269.828} C_DIS
LIN {X -0.069,Y -181.520,Z 1151.499,A 0.000,B 0.000,C 90.000,E1 269.828} C_DIS
LIN {X 0.031,Y -180.780,Z 1151.471,A 0.000,B 0.000,C 90.000,E1 264.723} C_DIS
LIN {X -0.075,Y -178.877,Z 1151.443,A 0.000,B 0.000,C 90.000,E1 259.690} C_DIS
LIN {X 0.001,Y -175.919,Z 1151.414,A 0.000,B 0.000,C 90.000,E1 254.574} C_DIS
LIN {X 0.057,Y -174.615,Z 1151.405,A 0.000,B 0.000,C 90.000,E1 252.851} C_DIS
LIN {X -0.016,Y -171.596,Z 1151.381,A 0.000,B 0.000,C 90.000,E1 248.592} C_DIS
LIN {X -0.027,Y -167.819,Z 1151.357,A 0.000,B 0.000,C 90.000,E1 244.280} C_DIS
LIN {X -0.010,Y -166.541,Z 1151.347,A 0.000,B 0.000,C 90.000,E1 242.538} C_DIS
LIN {X -0.099,Y -162.539,Z 1151.323,A 0.000,B 0.000,C 90.000,E1 238.201} C_DIS
LIN {X -0.039,Y -161.215,Z 1151.313,A 0.000,B 0.000,C 90.000,E1 236.421} C_DIS
LIN {X -0.003,Y -157.223,Z 1151.289,A 0.000,B 0.000,C 90.000,E1 231.984} C_DIS
LIN {X 0.020,Y -155.949,Z 1151.279,A 0.000,B 0.000,C 90.000,E1 230.194} C_DIS
LIN {X -0.021,Y -152.201,Z 1151.254,A 0.000,B 0.000,C 90.000,E1 225.729} C_DIS
LIN {X 0.000,Y -150.447,Z 1151.239,A 0.000,B 0.000,C 90.000,E1 223.014} C_DIS
LIN {X 0.027,Y -147.173,Z 1151.214,A 0.000,B 0.000,C 90.000,E1 218.463} C_DIS
LIN {X -0.006,Y -145.189,Z 1151.193,A 0.000,B 0.000,C 90.000,E1 214.818} C_DIS
LIN {X 0.028,Y -142.332,Z 1151.163,A 0.000,B 0.000,C 90.000,E1 209.283} C_DIS
LIN {X -0.042,Y -141.721,Z 1151.152,A 0.000,B 0.000,C 90.000,E1 207.462} C_DIS
LIN {X -0.060,Y -139.477,Z 1151.116,A 0.000,B 0.000,C 90.000,E1 200.972} C_DIS
LIN {X -0.071,Y -138.974,Z 1151.101,A 0.000,B 0.000,C 90.000,E1 198.181} C_DIS
LIN {X 0.051,Y -138.331,Z 1151.054,A 0.000,B 0.000,C 90.000,E1 189.726} C_DIS
LIN {X 0.054,Y -139.433,Z 1151.007,A 0.000,B 0.000,C 90.000,E1 181.318} C_DIS
LIN {X -0.006,Y -140.961,Z 1150.976,A 0.000,B 0.000,C 90.000,E1 175.755} C_DIS
LIN {X -0.056,Y -142.716,Z 1150.956,A 0.000,B 0.000,C 90.000,E1 172.064} C_DIS
LIN {X 0.043,Y -145.096,Z 1150.930,A 0.000,B 0.000,C 90.000,E1 167.409} C_DIS
LIN {X 0.038,Y -147.720,Z 1150.910,A 0.000,B 0.000,C 90.000,E1 163.740} C_DIS
LIN {X -0.020,Y -150.379,Z 1150.890,A 0.000,B 0.000,C 90.000,E1 160.115} C_DIS
LIN {X -0.003,Y -153.809,Z 1150.869,A 0.000,B 0.000,C 90.000,E1 156.485} C_DIS
LIN {X 0.056,Y -157.220,Z 1150.849,A 0.000,B 0.000,C 90.000,E1 152.871} C_DIS
LIN {X -0.003,Y -161.387,Z 1150.830,A 0.000,B 0.000,C 90.000,E1 149.331} C_DIS
LIN {X 0.008,Y -165.589,Z 1150.810,A 0.000,B 0.000,C 90.000,E1 145.801} C_DIS
LIN {X -0.005,Y -170.510,Z 1150.791,A 0.000,B 0.000,C 90.000,E1 142.316} C_DIS
LIN {X 0.039,Y -175.391,Z 1150.771,A 0.000,B 0.000,C 90.000,E1 138.852} C_DIS
LIN {X -0.099,Y -181.015,Z 1150.753,A 0.000,B 0.000,C 90.000,E1 135.486} C_DIS
LIN {X 0.025,Y -186.445,Z 1150.734,A 0.000,B 0.000,C 90.000,E1 132.081} C_DIS
LIN {X 0.094,Y -191.070,Z 1150.720,A 0.000,B 0.000,C 90.000,E1 129.564} C_DIS
LIN {X 0.015,Y -196.857,Z 1150.702,A 0.000,B 0.000,C 90.000,E1 126.297} C_DIS
LIN {X 0.052,Y -201.131,Z 1150.690,A 0.000,B 0.000,C 90.000,E1 124.119} C_DIS
LIN {X 0.033,Y -310.616,Z 1150.690,A 0.000,B 0.000,C 90.000,E1 124.119} C_DIS
LIN {X 0.009,Y -314.989,Z 1150.689,A 0.000,B 0.000,C 90.000,E1 123.992} C_DIS
LIN {X -0.015,Y -317.119,Z 1150.688,A 0.000,B 0.000,C 90.000,E1 123.865} C_DIS
LIN {X -0.061,Y -320.986,Z 1150.686,A 0.000,B 0.000,C 90.000,E1 123.499} C_DIS
LIN {X -0.086,Y -324.456,Z 1150.683,A 0.000,B 0.000,C 90.000,E1 122.959} C_DIS
LIN {X 0.000,Y -325.878,Z 1150.681,A 0.000,B 0.000,C 90.000,E1 122.625} C_DIS
LIN {X 0.123,Y -337.893,Z 1150.664,A 0.000,B 0.000,C 90.000,E1 119.461} C_DIS
LIN {X 0.099,Y -350.131,Z 1150.648,A 0.000,B 0.000,C 90.000,E1 116.693} C_DIS
LIN {X -0.047,Y -363.850,Z 1150.633,A 0.000,B 0.000,C 90.000,E1 114.003} C_DIS
LIN {X -0.046,Y -377.391,Z 1150.620,A 0.000,B 0.000,C 90.000,E1 111.642} C_DIS
LIN {X 0.023,Y -392.295,Z 1150.607,A 0.000,B 0.000,C 90.000,E1 109.322} C_DIS
LIN {X -0.166,Y -408.668,Z 1150.595,A 0.000,B 0.000,C 90.000,E1 107.094} C_DIS
LIN {X -0.191,Y -426.627,Z 1150.583,A 0.000,B 0.000,C 90.000,E1 104.898} C_DIS
LIN {X -0.181,Y -446.157,Z 1150.571,A 0.000,B 0.000,C 90.000,E1 102.771} C_DIS
LIN {X 0.012,Y -466.424,Z 1150.560,A 0.000,B 0.000,C 90.000,E1 100.782} C_DIS
LIN {X 0.018,Y -468.994,Z 1150.559,A 0.000,B 0.000,C 90.000,E1 100.546} C_DIS
LIN {X 0.027,Y -471.094,Z 1150.557,A 0.000,B 0.000,C 90.000,E1 100.310} C_DIS
LIN {X 0.036,Y -472.687,Z 1150.556,A 0.000,B 0.000,C 90.000,E1 100.074} C_DIS
LIN {X -0.188,Y -473.990,Z 1150.555,A 0.000,B 0.000,C 90.000,E1 99.849} C_DIS
LIN {X 0.137,Y -474.951,Z 1150.553,A 0.000,B 0.000,C 90.000,E1 99.557} C_DIS
LIN {X -0.210,Y -476.023,Z 1150.550,A 0.000,B 0.000,C 90.000,E1 99.095} C_DIS
LIN {X -0.007,Y -476.105,Z 1150.548,A 0.000,B 0.000,C 90.000,E1 98.568} C_DIS
LIN {X 0.128,Y -475.210,Z 1150.545,A 0.000,B 0.000,C 90.000,E1 98.049} C_DIS
LIN {X -0.204,Y -473.192,Z 1150.542,A 0.000,B 0.000,C 90.000,E1 97.587} C_DIS
LIN {X 0.127,Y -471.634,Z 1150.541,A 0.000,B 0.000,C 90.000,E1 97.296} C_DIS
LIN {X -0.205,Y -455.322,Z 1150.528,A 0.000,B 0.000,C 90.000,E1 95.049} C_DIS
LIN {X 0.093,Y -437.997,Z 1150.513,A 0.000,B 0.000,C 90.000,E1 92.407} C_DIS
LIN {X -0.023,Y -420.396,Z 1150.497,A 0.000,B 0.000,C 90.000,E1 89.484} C_DIS
LIN {X -0.065,Y -408.670,Z 1150.485,A 0.000,B 0.000,C 90.000,E1 87.306} C_DIS
LIN {X -0.049,Y -399.709,Z 1150.476,A 0.000,B 0.000,C 90.000,E1 85.641} C_DIS
LIN {X -0.092,Y -387.803,Z 1150.463,A 0.000,B 0.000,C 90.000,E1 83.394} C_DIS
LIN {X -0.009,Y -377.405,Z 1150.452,A 0.000,B 0.000,C 90.000,E1 81.376} C_DIS
LIN {X -0.031,Y -369.740,Z 1150.444,A 0.000,B 0.000,C 90.000,E1 79.926} C_DIS
LIN {X -0.127,Y -360.303,Z 1150.434,A 0.000,B 0.000,C 90.000,E1 78.173} C_DIS
LIN {X 0.033,Y -350.564,Z 1150.424,A 0.000,B 0.000,C 90.000,E1 76.353} C_DIS
LIN {X 0.092,Y -339.107,Z 1150.412,A 0.000,B 0.000,C 90.000,E1 74.212} C_DIS
LIN {X 0.138,Y -324.719,Z 1150.397,A 0.000,B 0.000,C 90.000,E1 71.402} C_DIS
LIN {X -0.065,Y -308.131,Z 1150.377,A 0.000,B 0.000,C 90.000,E1 67.922} C_DIS
LIN {X -0.086,Y -295.436,Z 1150.361,A 0.000,B 0.000,C 90.000,E1 64.973} C_DIS
LIN {X -0.039,Y -284.570,Z 1150.346,A 0.000,B 0.000,C 90.000,E1 62.281} C_DIS
LIN {X 0.001,Y -274.226,Z 1150.331,A 0.000,B 0.000,C 90.000,E1 59.537} C_DIS
LIN {X 0.158,Y -261.808,Z 1150.311,A 0.000,B 0.000,C 90.000,E1 56.008} C_DIS
LIN {X -0.078,Y -251.293,Z 1150.293,A 0.000,B 0.000,C 90.000,E1 52.844} C_DIS
LIN {X 0.011,Y -240.519,Z 1150.273,A 0.000,B 0.000,C 90.000,E1 49.175} C_DIS
LIN {X -0.123,Y -230.700,Z 1150.253,A 0.000,B 0.000,C 90.000,E1 45.486} C_DIS
LIN {X -0.066,Y -221.508,Z 1150.231,A 0.000,B 0.000,C 90.000,E1 41.676} C_DIS
LIN {X -0.073,Y -212.936,Z 1150.210,A 0.000,B 0.000,C 90.000,E1 37.810} C_DIS
LIN {X -0.051,Y -205.051,Z 1150.188,A 0.000,B 0.000,C 90.000,E1 33.865} C_DIS
LIN {X -0.096,Y -197.894,Z 1150.166,A 0.000,B 0.000,C 90.000,E1 29.873} C_DIS
LIN {X -0.064,Y -191.663,Z 1150.143,A 0.000,B 0.000,C 90.000,E1 25.796} C_DIS
LIN {X -0.029,Y -186.395,Z 1150.120,A 0.000,B 0.000,C 90.000,E1 21.663} C_DIS
LIN {X 0.083,Y -182.042,Z 1150.097,A 0.000,B 0.000,C 90.000,E1 17.457} C_DIS
LIN {X -0.086,Y -178.649,Z 1150.074,A 0.000,B 0.000,C 90.000,E1 13.300} C_DIS
LIN {X -0.076,Y -175.686,Z 1150.041,A 0.000,B 0.000,C 90.000,E1 7.352} C_DIS
LIN {X -0.057,Y -176.587,Z 1149.964,A 0.000,B 0.000,C 90.000,E1 353.571} C_DIS
LIN {X -0.040,Y -179.653,Z 1149.936,A 0.000,B 0.000,C 90.000,E1 348.465} C_DIS
LIN {X 0.064,Y -183.196,Z 1149.912,A 0.000,B 0.000,C 90.000,E1 344.212} C_DIS
LIN {X -0.044,Y -187.654,Z 1149.889,A 0.000,B 0.000,C 90.000,E1 340.061} C_DIS
LIN {X -0.049,Y -192.916,Z 1149.866,A 0.000,B 0.000,C 90.000,E1 335.921} C_DIS
LIN {X -0.013,Y -198.942,Z 1149.843,A 0.000,B 0.000,C 90.000,E1 331.820} C_DIS
LIN {X -0.003,Y -204.362,Z 1149.825,A 0.000,B 0.000,C 90.000,E1 328.584} C_DIS
LIN {X 0.003,Y -210.423,Z 1149.808,A 0.000,B 0.000,C 90.000,E1 325.388} C_DIS
LIN {X -0.127,Y -217.206,Z 1149.790,A 0.000,B 0.000,C 90.000,E1 322.271} C_DIS
LIN {X -0.025,Y -224.954,Z 1149.773,A 0.000,B 0.000,C 90.000,E1 319.138} C_DIS
LIN {X -0.094,Y -234.814,Z 1149.754,A 0.000,B 0.000,C 90.000,E1 315.729} C_DIS
LIN {X 0.132,Y -244.620,Z 1149.737,A 0.000,B 0.000,C 90.000,E1 312.690} C_DIS
LIN {X -0.044,Y -255.604,Z 1149.721,A 0.000,B 0.000,C 90.000,E1 309.806} C_DIS
LIN {X -0.071,Y -267.740,Z 1149.705,A 0.000,B 0.000,C 90.000,E1 306.950} C_DIS
LIN {X 0.059,Y -283.049,Z 1149.688,A 0.000,B 0.000,C 90.000,E1 303.785} C_DIS
LIN {X 0.025,Y -300.183,Z 1149.671,A 0.000,B 0.000,C 90.000,E1 300.747} C_DIS
LIN {X 0.070,Y -314.846,Z 1149.658,A 0.000,B 0.000,C 90.000,E1 298.437} C_DIS
LIN {X -0.092,Y -328.455,Z 1149.647,A 0.000,B 0.000,C 90.000,E1 296.539} C_DIS
LIN {X 0.137,Y -345.809,Z 1149.635,A 0.000,B 0.000,C 90.000,E1 294.335} C_DIS
LIN {X 0.130,Y -358.682,Z 1149.627,A 0.000,B 0.000,C 90.000,E1 292.898} C_DIS
LIN {X 0.055,Y -375.196,Z 1149.618,A 0.000,B 0.000,C 90.000,E1 291.280} C_DIS
LIN {X -0.190,Y -394.257,Z 1149.609,A 0.000,B 0.000,C 90.000,E1 289.577} C_DIS
LIN {X -0.179,Y -404.881,Z 1149.603,A 0.000,B 0.000,C 90.000,E1 288.598} C_DIS
LIN {X -0.129,Y -415.308,Z 1149.598,A 0.000,B 0.000,C 90.000,E1 287.583} C_DIS
LIN {X -0.118,Y -425.410,Z 1149.592,A 0.000,B 0.000,C 90.000,E1 286.551} C_DIS
LIN {X 0.112,Y -432.730,Z 1149.588,A 0.000,B 0.000,C 90.000,E1 285.733} C_DIS
LIN {X -0.059,Y -439.632,Z 1149.583,A 0.000,B 0.000,C 90.000,E1 284.954} C_DIS
LIN {X 0.248,Y -445.915,Z 1149.579,A 0.000,B 0.000,C 90.000,E1 284.120} C_DIS
LIN {X 0.076,Y -451.403,Z 1149.574,A 0.000,B 0.000,C 90.000,E1 283.355} C_DIS
LIN {X -0.054,Y -456.238,Z 1149.570,A 0.000,B 0.000,C 90.000,E1 282.591} C_DIS
LIN {X -0.140,Y -460.440,Z 1149.566,A 0.000,B 0.000,C 90.000,E1 281.827} C_DIS
LIN {X 0.170,Y -464.051,Z 1149.561,A 0.000,B 0.000,C 90.000,E1 281.018} C_DIS
LIN {X -0.150,Y -466.223,Z 1149.558,A 0.000,B 0.000,C 90.000,E1 280.546} C_DIS
LIN {X -0.003,Y -468.192,Z 1149.556,A 0.000,B 0.000,C 90.000,E1 280.018} C_DIS
LIN {X 0.233,Y -471.528,Z 1149.550,A 0.000,B 0.000,C 90.000,E1 278.973} C_DIS
LIN {X -0.136,Y -472.819,Z 1149.547,A 0.000,B 0.000,C 90.000,E1 278.511} C_DIS
LIN {X -0.025,Y -473.828,Z 1149.544,A 0.000,B 0.000,C 90.000,E1 277.992} C_DIS
LIN {X 0.095,Y -474.558,Z 1149.542,A 0.000,B 0.000,C 90.000,E1 277.473} C_DIS
LIN {X -0.191,Y -474.941,Z 1149.539,A 0.000,B 0.000,C 90.000,E1 277.004} C_DIS
LIN {X -0.063,Y -474.924,Z 1149.536,A 0.000,B 0.000,C 90.000,E1 276.486} C_DIS
LIN {X 0.067,Y -474.492,Z 1149.533,A 0.000,B 0.000,C 90.000,E1 275.967} C_DIS
LIN {X 0.150,Y -473.642,Z 1149.530,A 0.000,B 0.000,C 90.000,E1 275.454} C_DIS
LIN {X -0.191,Y -472.331,Z 1149.528,A 0.000,B 0.000,C 90.000,E1 274.992} C_DIS
LIN {X -0.068,Y -470.561,Z 1149.525,A 0.000,B 0.000,C 90.000,E1 274.473} C_DIS
LIN {X 0.044,Y -468.253,Z 1149.522,A 0.000,B 0.000,C 90.000,E1 273.955} C_DIS
LIN {X 0.107,Y -465.342,Z 1149.519,A 0.000,B 0.000,C 90.000,E1 273.440} C_DIS
LIN {X 0.183,Y -461.620,Z 1149.516,A 0.000,B 0.000,C 90.000,E1 272.922} C_DIS
LIN {X 0.214,Y -456.801,Z 1149.514,A 0.000,B 0.000,C 90.000,E1 272.407} C_DIS
LIN {X 0.041,Y -454.006,Z 1149.512,A 0.000,B 0.000,C 90.000,E1 272.178} C_DIS
LIN {X -0.129,Y -450.850,Z 1149.511,A 0.000,B 0.000,C 90.000,E1 271.949} C_DIS
LIN {X 0.099,Y -444.244,Z 1149.508,A 0.000,B 0.000,C 90.000,E1 271.489} C_DIS
LIN {X 0.012,Y -437.470,Z 1149.506,A 0.000,B 0.000,C 90.000,E1 271.146} C_DIS
LIN {X -0.090,Y -430.385,Z 1149.505,A 0.000,B 0.000,C 90.000,E1 270.859} C_DIS
LIN {X -0.208,Y -423.245,Z 1149.503,A 0.000,B 0.000,C 90.000,E1 270.630} C_DIS
LIN {X 0.189,Y -412.613,Z 1149.502,A 0.000,B 0.000,C 90.000,E1 270.286} C_DIS
LIN {X 0.156,Y -401.604,Z 1149.500,A 0.000,B 0.000,C 90.000,E1 270.057} C_DIS
LIN {X 0.122,Y -390.632,Z 1149.500,A 0.000,B 0.000,C 90.000,E1 269.885} C_DIS
LIN {X 0.017,Y -382.537,Z 1149.499,A 0.000,B 0.000,C 90.000,E1 269.828} C_DIS
LIN {X -0.180,Y -373.965,Z 1149.499,A 0.000,B 0.000,C 90.000,E1 269.828} C_DIS
LIN {X 0.063,Y -181.515,Z 1149.499,A 0.000,B 0.000,C 90.000,E1 269.771} C_DIS
LIN {X -0.076,Y -180.908,Z 1149.475,A 0.000,B 0.000,C 90.000,E1 265.584} C_DIS
LIN {X -0.018,Y -180.774,Z 1149.471,A 0.000,B 0.000,C 90.000,E1 264.723} C_DIS
LIN {X 0.053,Y -178.870,Z 1149.443,A 0.000,B 0.000,C 90.000,E1 259.634} C_DIS
LIN {X -0.046,Y -175.913,Z 1149.414,A 0.000,B 0.000,C 90.000,E1 254.574} C_DIS
LIN {X 0.009,Y -174.602,Z 1149.405,A 0.000,B 0.000,C 90.000,E1 252.851} C_DIS
LIN {X -0.064,Y -171.584,Z 1149.381,A 0.000,B 0.000,C 90.000,E1 248.592} C_DIS
LIN {X -0.074,Y -167.807,Z 1149.357,A 0.000,B 0.000,C 90.000,E1 244.280} C_DIS
LIN {X -0.056,Y -166.527,Z 1149.347,A 0.000,B 0.000,C 90.000,E1 242.538} C_DIS
LIN {X 0.079,Y -162.526,Z 1149.323,A 0.000,B 0.000,C 90.000,E1 238.122} C_DIS
LIN {X 0.050,Y -161.201,Z 1149.313,A 0.000,B 0.000,C 90.000,E1 236.373} C_DIS
LIN {X -0.048,Y -157.210,Z 1149.289,A 0.000,B 0.000,C 90.000,E1 231.984} C_DIS
LIN {X -0.025,Y -155.937,Z 1149.279,A 0.000,B 0.000,C 90.000,E1 230.194} C_DIS
LIN {X -0.065,Y -152.189,Z 1149.254,A 0.000,B 0.000,C 90.000,E1 225.729} C_DIS
LIN {X -0.044,Y -150.436,Z 1149.239,A 0.000,B 0.000,C 90.000,E1 223.014} C_DIS
LIN {X -0.016,Y -147.163,Z 1149.214,A 0.000,B 0.000,C 90.000,E1 218.463} C_DIS
LIN {X -0.049,Y -145.179,Z 1149.193,A 0.000,B 0.000,C 90.000,E1 214.818} C_DIS
LIN {X -0.014,Y -142.325,Z 1149.163,A 0.000,B 0.000,C 90.000,E1 209.283} C_DIS
LIN {X -0.019,Y -141.715,Z 1149.152,A 0.000,B 0.000,C 90.000,E1 207.436} C_DIS
LIN {X 0.029,Y -139.474,Z 1149.116,A 0.000,B 0.000,C 90.000,E1 200.918} C_DIS
LIN {X 0.020,Y -138.969,Z 1149.101,A 0.000,B 0.000,C 90.000,E1 198.127} C_DIS
LIN {X 0.009,Y -138.330,Z 1149.054,A 0.000,B 0.000,C 90.000,E1 189.726} C_DIS
LIN {X 0.012,Y -139.437,Z 1149.007,A 0.000,B 0.000,C 90.000,E1 181.318} C_DIS
LIN {X -0.049,Y -140.968,Z 1148.976,A 0.000,B 0.000,C 90.000,E1 175.755} C_DIS
LIN {X 0.043,Y -142.723,Z 1148.956,A 0.000,B 0.000,C 90.000,E1 172.008} C_DIS
LIN {X 0.001,Y -145.106,Z 1148.930,A 0.000,B 0.000,C 90.000,E1 167.409} C_DIS
LIN {X -0.005,Y -147.731,Z 1148.910,A 0.000,B 0.000,C 90.000,E1 163.740} C_DIS
LIN {X 0.077,Y -150.393,Z 1148.889,A 0.000,B 0.000,C 90.000,E1 160.061} C_DIS
LIN {X -0.047,Y -153.827,Z 1148.869,A 0.000,B 0.000,C 90.000,E1 156.485} C_DIS
LIN {X 0.011,Y -157.238,Z 1148.849,A 0.000,B 0.000,C 90.000,E1 152.871} C_DIS
LIN {X -0.048,Y -161.408,Z 1148.829,A 0.000,B 0.000,C 90.000,E1 149.331} C_DIS
LIN {X -0.039,Y -165.610,Z 1148.810,A 0.000,B 0.000,C 90.000,E1 145.801} C_DIS
LIN {X 0.082,Y -170.536,Z 1148.791,A 0.000,B 0.000,C 90.000,E1 142.271} C_DIS
LIN {X -0.009,Y -175.414,Z 1148.771,A 0.000,B 0.000,C 90.000,E1 138.852} C_DIS
LIN {X -0.019,Y -181.038,Z 1148.752,A 0.000,B 0.000,C 90.000,E1 135.445} C_DIS
LIN {X -0.025,Y -186.472,Z 1148.734,A 0.000,B 0.000,C 90.000,E1 132.081} C_DIS
LIN {X 0.043,Y -191.094,Z 1148.720,A 0.000,B 0.000,C 90.000,E1 129.564} C_DIS
LIN {X -0.036,Y -196.887,Z 1148.702,A 0.000,B 0.000,C 90.000,E1 126.297} C_DIS
LIN {X -0.001,Y -201.157,Z 1148.690,A 0.000,B 0.000,C 90.000,E1 124.119} C_DIS
LIN {X -0.048,Y -310.099,Z 1148.689,A 0.000,B 0.000,C 90.000,E1 124.119} C_DIS
LIN {X -0.073,Y -314.955,Z 1148.689,A 0.000,B 0.000,C 90.000,E1 123.992} C_DIS
LIN {X 0.079,Y -317.111,Z 1148.688,A 0.000,B 0.000,C 90.000,E1 123.833} C_DIS
LIN {X -0.123,Y -320.968,Z 1148.686,A 0.000,B 0.000,C 90.000,E1 123.499} C_DIS
LIN {X -0.128,Y -324.446,Z 1148.683,A 0.000,B 0.000,C 90.000,E1 122.959} C_DIS
LIN {X -0.042,Y -325.880,Z 1148.681,A 0.000,B 0.000,C 90.000,E1 122.625} C_DIS
LIN {X 0.079,Y -337.902,Z 1148.664,A 0.000,B 0.000,C 90.000,E1 119.461} C_DIS
LIN {X 0.055,Y -350.143,Z 1148.648,A 0.000,B 0.000,C 90.000,E1 116.693} C_DIS
LIN {X -0.093,Y -363.865,Z 1148.633,A 0.000,B 0.000,C 90.000,E1 114.003} C_DIS
LIN {X -0.092,Y -377.410,Z 1148.620,A 0.000,B 0.000,C 90.000,E1 111.642} C_DIS
LIN {X -0.026,Y -392.318,Z 1148.607,A 0.000,B 0.000,C 90.000,E1 109.322} C_DIS
LIN {X 0.174,Y -408.697,Z 1148.595,A 0.000,B 0.000,C 90.000,E1 107.040} C_DIS
LIN {X -0.133,Y -426.660,Z 1148.583,A 0.000,B 0.000,C 90.000,E1 104.883} C_DIS
LIN {X -0.234,Y -446.193,Z 1148.571,A 0.000,B 0.000,C 90.000,E1 102.771} C_DIS
LIN {X -0.033,Y -469.027,Z 1148.559,A 0.000,B 0.000,C 90.000,E1 100.546} C_DIS
LIN {X -0.026,Y -471.110,Z 1148.557,A 0.000,B 0.000,C 90.000,E1 100.310} C_DIS
LIN {X -0.020,Y -472.689,Z 1148.556,A 0.000,B 0.000,C 90.000,E1 100.074} C_DIS
LIN {X -0.244,Y -473.979,Z 1148.555,A 0.000,B 0.000,C 90.000,E1 99.849} C_DIS
LIN {X 0.082,Y -474.931,Z 1148.553,A 0.000,B 0.000,C 90.000,E1 99.557} C_DIS
LIN {X -0.191,Y -475.986,Z 1148.550,A 0.000,B 0.000,C 90.000,E1 99.086} C_DIS
LIN {X -0.064,Y -476.052,Z 1148.548,A 0.000,B 0.000,C 90.000,E1 98.568} C_DIS
LIN {X 0.072,Y -475.141,Z 1148.545,A 0.000,B 0.000,C 90.000,E1 98.049} C_DIS
LIN {X 0.209,Y -473.102,Z 1148.542,A 0.000,B 0.000,C 90.000,E1 97.530} C_DIS
LIN {X 0.071,Y -471.530,Z 1148.541,A 0.000,B 0.000,C 90.000,E1 97.296} C_DIS
LIN {X 0.191,Y -455.187,Z 1148.528,A 0.000,B 0.000,C 90.000,E1 94.992} C_DIS
LIN {X 0.034,Y -437.882,Z 1148.513,A 0.000,B 0.000,C 90.000,E1 92.407} C_DIS
LIN {X -0.083,Y -420.281,Z 1148.497,A 0.000,B 0.000,C 90.000,E1 89.484} C_DIS
LIN {X -0.126,Y -408.559,Z 1148.485,A 0.000,B 0.000,C 90.000,E1 87.306} C_DIS
LIN {X -0.110,Y -399.579,Z 1148.476,A 0.000,B 0.000,C 90.000,E1 85.641} C_DIS
LIN {X -0.153,Y -386.178,Z 1148.462,A 0.000,B 0.000,C 90.000,E1 83.109} C_DIS
LIN {X -0.058,Y -375.770,Z 1148.450,A 0.000,B 0.000,C 90.000,E1 81.084} C_DIS
LIN {X -0.110,Y -366.477,Z 1148.441,A 0.000,B 0.000,C 90.000,E1 79.342} C_DIS
LIN {X 0.165,Y -356.934,Z 1148.431,A 0.000,B 0.000,C 90.000,E1 77.521} C_DIS
LIN {X -0.148,Y -345.473,Z 1148.419,A 0.000,B 0.000,C 90.000,E1 75.463} C_DIS
LIN {X 0.110,Y -332.442,Z 1148.405,A 0.000,B 0.000,C 90.000,E1 72.960} C_DIS
LIN {X 0.069,Y -318.330,Z 1148.390,A 0.000,B 0.000,C 90.000,E1 70.134} C_DIS
LIN {X -0.016,Y -303.670,Z 1148.372,A 0.000,B 0.000,C 90.000,E1 66.922} C_DIS
LIN {X -0.029,Y -291.160,Z 1148.355,A 0.000,B 0.000,C 90.000,E1 63.948} C_DIS
LIN {X 0.074,Y -277.877,Z 1148.336,A 0.000,B 0.000,C 90.000,E1 60.539} C_DIS
LIN {X -0.019,Y -267.707,Z 1148.321,A 0.000,B 0.000,C 90.000,E1 57.788} C_DIS
LIN {X -0.027,Y -256.852,Z 1148.303,A 0.000,B 0.000,C 90.000,E1 54.609} C_DIS
LIN {X -0.087,Y -246.637,Z 1148.285,A 0.000,B 0.000,C 90.000,E1 51.376} C_DIS
LIN {X 0.003,Y -236.276,Z 1148.265,A 0.000,B 0.000,C 90.000,E1 47.676} C_DIS
LIN {X 0.017,Y -228.608,Z 1148.248,A 0.000,B 0.000,C 90.000,E1 44.676} C_DIS
LIN {X 0.018,Y -219.506,Z 1148.227,A 0.000,B 0.000,C 90.000,E1 40.862} C_DIS
LIN {X -0.053,Y -211.022,Z 1148.205,A 0.000,B 0.000,C 90.000,E1 36.996} C_DIS
LIN {X -0.037,Y -204.752,Z 1148.188,A 0.000,B 0.000,C 90.000,E1 33.833} C_DIS
LIN {X 0.067,Y -197.587,Z 1148.166,A 0.000,B 0.000,C 90.000,E1 29.795} C_DIS
LIN {X -0.009,Y -192.524,Z 1148.148,A 0.000,B 0.000,C 90.000,E1 26.565} C_DIS
LIN {X -0.047,Y -187.048,Z 1148.125,A 0.000,B 0.000,C 90.000,E1 22.461} C_DIS
LIN {X -0.026,Y -182.507,Z 1148.102,A 0.000,B 0.000,C 90.000,E1 18.290} C_DIS
LIN {X 0.035,Y -178.905,Z 1148.078,A 0.000,B 0.000,C 90.000,E1 14.064} C_DIS
LIN {X 0.038,Y -176.029,Z 1148.050,A 0.000,B 0.000,C 90.000,E1 8.973} C_DIS
LIN {X -0.071,Y -176.255,Z 1147.964,A 0.000,B 0.000,C 90.000,E1 353.571} C_DIS
LIN {X -0.066,Y -179.295,Z 1147.936,A 0.000,B 0.000,C 90.000,E1 348.465} C_DIS
LIN {X 0.026,Y -182.837,Z 1147.912,A 0.000,B 0.000,C 90.000,E1 344.212} C_DIS
LIN {X -0.094,Y -187.282,Z 1147.889,A 0.000,B 0.000,C 90.000,E1 340.061} C_DIS
LIN {X 0.065,Y -192.531,Z 1147.866,A 0.000,B 0.000,C 90.000,E1 335.869} C_DIS
LIN {X -0.023,Y -197.292,Z 1147.848,A 0.000,B 0.000,C 90.000,E1 332.615} C_DIS
LIN {X 0.115,Y -202.599,Z 1147.830,A 0.000,B 0.000,C 90.000,E1 329.331} C_DIS
LIN {X -0.035,Y -208.515,Z 1147.812,A 0.000,B 0.000,C 90.000,E1 326.167} C_DIS
LIN {X -0.045,Y -215.148,Z 1147.794,A 0.000,B 0.000,C 90.000,E1 323.004} C_DIS
LIN {X -0.139,Y -222.686,Z 1147.777,A 0.000,B 0.000,C 90.000,E1 319.908} C_DIS
LIN {X -0.064,Y -231.213,Z 1147.760,A 0.000,B 0.000,C 90.000,E1 316.824} C_DIS
LIN {X 0.065,Y -240.652,Z 1147.743,A 0.000,B 0.000,C 90.000,E1 313.785} C_DIS
LIN {X -0.050,Y -251.218,Z 1147.727,A 0.000,B 0.000,C 90.000,E1 310.862} C_DIS
LIN {X 0.025,Y -264.493,Z 1147.709,A 0.000,B 0.000,C 90.000,E1 307.604} C_DIS
LIN {X -0.004,Y -279.548,Z 1147.691,A 0.000,B 0.000,C 90.000,E1 304.452} C_DIS
LIN {X -0.107,Y -290.525,Z 1147.680,A 0.000,B 0.000,C 90.000,E1 302.418} C_DIS
LIN {X -0.086,Y -308.480,Z 1147.663,A 0.000,B 0.000,C 90.000,E1 299.411} C_DIS
LIN {X 0.069,Y -326.218,Z 1147.649,A 0.000,B 0.000,C 90.000,E1 296.796} C_DIS
LIN {X 0.168,Y -340.938,Z 1147.638,A 0.000,B 0.000,C 90.000,E1 294.899} C_DIS
LIN {X 0.193,Y -353.903,Z 1147.630,A 0.000,B 0.000,C 90.000,E1 293.387} C_DIS
LIN {X -0.077,Y -367.476,Z 1147.622,A 0.000,B 0.000,C 90.000,E1 292.025} C_DIS
LIN {X 0.185,Y -389.502,Z 1147.611,A 0.000,B 0.000,C 90.000,E1 289.939} C_DIS
LIN {X 0.186,Y -400.327,Z 1147.605,A 0.000,B 0.000,C 90.000,E1 288.960} C_DIS
LIN {X -0.075,Y -410.865,Z 1147.600,A 0.000,B 0.000,C 90.000,E1 288.000} C_DIS
LIN {X -0.110,Y -421.129,Z 1147.594,A 0.000,B 0.000,C 90.000,E1 286.985} C_DIS
LIN {X -0.125,Y -428.630,Z 1147.590,A 0.000,B 0.000,C 90.000,E1 286.205} C_DIS
LIN {X 0.114,Y -435.881,Z 1147.585,A 0.000,B 0.000,C 90.000,E1 285.371} C_DIS
LIN {X -0.040,Y -442.539,Z 1147.581,A 0.000,B 0.000,C 90.000,E1 284.592} C_DIS
LIN {X 0.191,Y -448.488,Z 1147.577,A 0.000,B 0.000,C 90.000,E1 283.772} C_DIS
LIN {X 0.038,Y -453.720,Z 1147.572,A 0.000,B 0.000,C 90.000,E1 283.008} C_DIS
LIN {X -0.065,Y -458.303,Z 1147.568,A 0.000,B 0.000,C 90.000,E1 282.243} C_DIS
LIN {X -0.135,Y -462.245,Z 1147.564,A 0.000,B 0.000,C 90.000,E1 281.478} C_DIS
LIN {X 0.041,Y -466.740,Z 1147.558,A 0.000,B 0.000,C 90.000,E1 280.433} C_DIS
LIN {X 0.192,Y -468.673,Z 1147.555,A 0.000,B 0.000,C 90.000,E1 279.905} C_DIS
LIN {X -0.117,Y -470.421,Z 1147.552,A 0.000,B 0.000,C 90.000,E1 279.434} C_DIS
LIN {X -0.028,Y -471.968,Z 1147.550,A 0.000,B 0.000,C 90.000,E1 278.916} C_DIS
LIN {X 0.075,Y -473.222,Z 1147.547,A 0.000,B 0.000,C 90.000,E1 278.398} C_DIS
LIN {X 0.254,Y -474.206,Z 1147.544,A 0.000,B 0.000,C 90.000,E1 277.871} C_DIS
LIN {X -0.096,Y -474.868,Z 1147.541,A 0.000,B 0.000,C 90.000,E1 277.409} C_DIS
LIN {X 0.029,Y -475.183,Z 1147.538,A 0.000,B 0.000,C 90.000,E1 276.891} C_DIS
LIN {X 0.160,Y -475.102,Z 1147.536,A 0.000,B 0.000,C 90.000,E1 276.372} C_DIS
LIN {X -0.180,Y -474.642,Z 1147.533,A 0.000,B 0.000,C 90.000,E1 275.910} C_DIS
LIN {X -0.048,Y -473.746,Z 1147.530,A 0.000,B 0.000,C 90.000,E1 275.391} C_DIS
LIN {X 0.038,Y -472.366,Z 1147.527,A 0.000,B 0.000,C 90.000,E1 274.878} C_DIS
LIN {X 0.161,Y -470.560,Z 1147.524,A 0.000,B 0.000,C 90.000,E1 274.359} C_DIS
LIN {X -0.196,Y -468.195,Z 1147.521,A 0.000,B 0.000,C 90.000,E1 273.898} C_DIS
LIN {X -0.130,Y -465.201,Z 1147.519,A 0.000,B 0.000,C 90.000,E1 273.383} C_DIS
LIN {X -0.053,Y -461.351,Z 1147.516,A 0.000,B 0.000,C 90.000,E1 272.865} C_DIS
LIN {X -0.019,Y -456.446,Z 1147.513,A 0.000,B 0.000,C 90.000,E1 272.350} C_DIS
LIN {X 0.140,Y -450.371,Z 1147.510,A 0.000,B 0.000,C 90.000,E1 271.835} C_DIS
LIN {X -0.162,Y -447.240,Z 1147.509,A 0.000,B 0.000,C 90.000,E1 271.661} C_DIS
LIN {X -0.029,Y -440.460,Z 1147.507,A 0.000,B 0.000,C 90.000,E1 271.260} C_DIS
LIN {X 0.171,Y -433.548,Z 1147.505,A 0.000,B 0.000,C 90.000,E1 270.917} C_DIS
LIN {X -0.115,Y -426.424,Z 1147.504,A 0.000,B 0.000,C 90.000,E1 270.688} C_DIS
LIN {X -0.051,Y -419.236,Z 1147.503,A 0.000,B 0.000,C 90.000,E1 270.458} C_DIS
LIN {X 0.109,Y -408.492,Z 1147.501,A 0.000,B 0.000,C 90.000,E1 270.172} C_DIS
LIN {X -0.149,Y -397.584,Z 1147.500,A 0.000,B 0.000,C 90.000,E1 270.000} C_DIS
LIN {X -0.150,Y -389.305,Z 1147.499,A 0.000,B 0.000,C 90.000,E1 269.885} C_DIS
LIN {X 0.149,Y -377.857,Z 1147.499,A 0.000,B 0.000,C 90.000,E1 269.771} C_DIS
LIN {X 0.094,Y -373.755,Z 1147.499,A 0.000,B 0.000,C 90.000,E1 269.771} C_DIS
LIN {X 0.019,Y -181.511,Z 1147.499,A 0.000,B 0.000,C 90.000,E1 269.771} C_DIS
LIN {X 0.019,Y -180.908,Z 1147.475,A 0.000,B 0.000,C 90.000,E1 265.527} C_DIS
LIN {X 0.077,Y -180.764,Z 1147.470,A 0.000,B 0.000,C 90.000,E1 264.666} C_DIS
LIN {X -0.032,Y -178.857,Z 1147.442,A 0.000,B 0.000,C 90.000,E1 259.634} C_DIS
LIN {X 0.039,Y -175.901,Z 1147.414,A 0.000,B 0.000,C 90.000,E1 254.519} C_DIS
LIN {X -0.023,Y -174.579,Z 1147.405,A 0.000,B 0.000,C 90.000,E1 252.834} C_DIS
LIN {X 0.013,Y -171.562,Z 1147.381,A 0.000,B 0.000,C 90.000,E1 248.539} C_DIS
LIN {X -0.005,Y -167.786,Z 1147.357,A 0.000,B 0.000,C 90.000,E1 244.229} C_DIS
LIN {X 0.010,Y -166.501,Z 1147.347,A 0.000,B 0.000,C 90.000,E1 242.487} C_DIS
LIN {X 0.006,Y -163.210,Z 1147.328,A 0.000,B 0.000,C 90.000,E1 238.997} C_DIS
LIN {X -0.029,Y -161.174,Z 1147.313,A 0.000,B 0.000,C 90.000,E1 236.373} C_DIS
LIN {X 0.095,Y -157.188,Z 1147.289,A 0.000,B 0.000,C 90.000,E1 231.904} C_DIS
LIN {X 0.017,Y -155.917,Z 1147.279,A 0.000,B 0.000,C 90.000,E1 230.150} C_DIS
LIN {X 0.073,Y -152.169,Z 1147.254,A 0.000,B 0.000,C 90.000,E1 225.648} C_DIS
LIN {X -0.017,Y -150.417,Z 1147.239,A 0.000,B 0.000,C 90.000,E1 222.975} C_DIS
LIN {X -0.091,Y -147.145,Z 1147.214,A 0.000,B 0.000,C 90.000,E1 218.463} C_DIS
LIN {X 0.021,Y -145.704,Z 1147.198,A 0.000,B 0.000,C 90.000,E1 215.678} C_DIS
LIN {X 0.028,Y -143.086,Z 1147.173,A 0.000,B 0.000,C 90.000,E1 211.082} C_DIS
LIN {X 0.033,Y -141.704,Z 1147.152,A 0.000,B 0.000,C 90.000,E1 207.385} C_DIS
LIN {X -0.044,Y -139.469,Z 1147.116,A 0.000,B 0.000,C 90.000,E1 200.918} C_DIS
LIN {X 0.010,Y -139.200,Z 1147.106,A 0.000,B 0.000,C 90.000,E1 199.033} C_DIS
LIN {X 0.073,Y -138.327,Z 1147.054,A 0.000,B 0.000,C 90.000,E1 189.670} C_DIS
LIN {X -0.061,Y -139.443,Z 1147.007,A 0.000,B 0.000,C 90.000,E1 181.318} C_DIS
LIN {X 0.018,Y -140.980,Z 1146.976,A 0.000,B 0.000,C 90.000,E1 175.698} C_DIS
LIN {X -0.031,Y -142.736,Z 1146.956,A 0.000,B 0.000,C 90.000,E1 172.008} C_DIS
LIN {X -0.075,Y -145.125,Z 1146.930,A 0.000,B 0.000,C 90.000,E1 167.409} C_DIS
LIN {X 0.061,Y -147.749,Z 1146.910,A 0.000,B 0.000,C 90.000,E1 163.685} C_DIS
LIN {X 0.000,Y -150.417,Z 1146.889,A 0.000,B 0.000,C 90.000,E1 160.061} C_DIS
LIN {X 0.016,Y -153.857,Z 1146.869,A 0.000,B 0.000,C 90.000,E1 156.433} C_DIS
LIN {X -0.068,Y -157.268,Z 1146.849,A 0.000,B 0.000,C 90.000,E1 152.871} C_DIS
LIN {X 0.010,Y -161.445,Z 1146.829,A 0.000,B 0.000,C 90.000,E1 149.282} C_DIS
LIN {X 0.017,Y -165.645,Z 1146.810,A 0.000,B 0.000,C 90.000,E1 145.754} C_DIS
LIN {X -0.001,Y -170.579,Z 1146.790,A 0.000,B 0.000,C 90.000,E1 142.271} C_DIS
LIN {X -0.093,Y -175.456,Z 1146.771,A 0.000,B 0.000,C 90.000,E1 138.852} C_DIS
LIN {X 0.022,Y -181.079,Z 1146.752,A 0.000,B 0.000,C 90.000,E1 135.405} C_DIS
LIN {X 0.012,Y -186.520,Z 1146.734,A 0.000,B 0.000,C 90.000,E1 132.043} C_DIS
LIN {X -0.046,Y -191.137,Z 1146.720,A 0.000,B 0.000,C 90.000,E1 129.564} C_DIS
LIN {X 0.032,Y -196.937,Z 1146.701,A 0.000,B 0.000,C 90.000,E1 126.251} C_DIS
LIN {X -0.060,Y -201.185,Z 1146.689,A 0.000,B 0.000,C 90.000,E1 124.119} C_DIS
LIN {X -0.139,Y -310.766,Z 1146.689,A 0.000,B 0.000,C 90.000,E1 124.119} C_DIS
LIN {X -0.064,Y -317.325,Z 1146.688,A 0.000,B 0.000,C 90.000,E1 123.833} C_DIS
LIN {X -0.190,Y -320.316,Z 1146.686,A 0.000,B 0.000,C 90.000,E1 123.579} C_DIS
LIN {X -0.112,Y -323.972,Z 1146.683,A 0.000,B 0.000,C 90.000,E1 123.038} C_DIS
LIN {X 0.148,Y -325.515,Z 1146.682,A 0.000,B 0.000,C 90.000,E1 122.673} C_DIS
LIN {X -0.073,Y -338.840,Z 1146.662,A 0.000,B 0.000,C 90.000,E1 119.255} C_DIS
LIN {X -0.076,Y -351.195,Z 1146.647,A 0.000,B 0.000,C 90.000,E1 116.488} C_DIS
LIN {X -0.027,Y -365.050,Z 1146.632,A 0.000,B 0.000,C 90.000,E1 113.770} C_DIS
LIN {X 0.016,Y -378.717,Z 1146.619,A 0.000,B 0.000,C 90.000,E1 111.408} C_DIS
LIN {X 0.128,Y -393.758,Z 1146.606,A 0.000,B 0.000,C 90.000,E1 109.087} C_DIS
LIN {X -0.017,Y -410.279,Z 1146.594,A 0.000,B 0.000,C 90.000,E1 106.858} C_DIS
LIN {X 0.010,Y -428.398,Z 1146.581,A 0.000,B 0.000,C 90.000,E1 104.662} C_DIS
LIN {X 0.115,Y -448.042,Z 1146.570,A 0.000,B 0.000,C 90.000,E1 102.535} C_DIS
LIN {X -0.008,Y -468.362,Z 1146.559,A 0.000,B 0.000,C 90.000,E1 100.602} C_DIS
LIN {X 0.032,Y -470.570,Z 1146.558,A 0.000,B 0.000,C 90.000,E1 100.366} C_DIS
LIN {X -0.013,Y -472.238,Z 1146.556,A 0.000,B 0.000,C 90.000,E1 100.141} C_DIS
LIN {X -0.155,Y -473.628,Z 1146.555,A 0.000,B 0.000,C 90.000,E1 99.905} C_DIS
LIN {X 0.168,Y -474.661,Z 1146.553,A 0.000,B 0.000,C 90.000,E1 99.613} C_DIS
LIN {X -0.182,Y -475.854,Z 1146.551,A 0.000,B 0.000,C 90.000,E1 99.151} C_DIS
LIN {X 0.018,Y -476.042,Z 1146.548,A 0.000,B 0.000,C 90.000,E1 98.624} C_DIS
LIN {X 0.151,Y -475.260,Z 1146.545,A 0.000,B 0.000,C 90.000,E1 98.106} C_DIS
LIN {X -0.182,Y -473.383,Z 1146.542,A 0.000,B 0.000,C 90.000,E1 97.644} C_DIS
LIN {X 0.150,Y -471.922,Z 1146.541,A 0.000,B 0.000,C 90.000,E1 97.352} C_DIS
LIN {X -0.179,Y -455.574,Z 1146.528,A 0.000,B 0.000,C 90.000,E1 95.106} C_DIS
LIN {X 0.124,Y -438.247,Z 1146.514,A 0.000,B 0.000,C 90.000,E1 92.465} C_DIS
LIN {X 0.131,Y -419.105,Z 1146.496,A 0.000,B 0.000,C 90.000,E1 89.255} C_DIS
LIN {X -0.024,Y -408.875,Z 1146.485,A 0.000,B 0.000,C 90.000,E1 87.364} C_DIS
LIN {X -0.004,Y -399.886,Z 1146.476,A 0.000,B 0.000,C 90.000,E1 85.698} C_DIS
LIN {X -0.040,Y -386.485,Z 1146.462,A 0.000,B 0.000,C 90.000,E1 83.166} C_DIS
LIN {X 0.044,Y -377.570,Z 1146.452,A 0.000,B 0.000,C 90.000,E1 81.432} C_DIS
LIN {X 0.023,Y -368.375,Z 1146.443,A 0.000,B 0.000,C 90.000,E1 79.690} C_DIS
LIN {X -0.096,Y -358.856,Z 1146.433,A 0.000,B 0.000,C 90.000,E1 77.937} C_DIS
LIN {X 0.037,Y -349.042,Z 1146.423,A 0.000,B 0.000,C 90.000,E1 76.117} C_DIS
LIN {X -0.043,Y -335.947,Z 1146.409,A 0.000,B 0.000,C 90.000,E1 73.685} C_DIS
LIN {X 0.016,Y -321.671,Z 1146.394,A 0.000,B 0.000,C 90.000,E1 70.859} C_DIS
LIN {X -0.167,Y -305.321,Z 1146.374,A 0.000,B 0.000,C 90.000,E1 67.358} C_DIS
LIN {X -0.128,Y -294.124,Z 1146.359,A 0.000,B 0.000,C 90.000,E1 64.717} C_DIS
LIN {X -0.111,Y -283.275,Z 1146.344,A 0.000,B 0.000,C 90.000,E1 62.025} C_DIS
LIN {X 0.037,Y -272.926,Z 1146.329,A 0.000,B 0.000,C 90.000,E1 59.253} C_DIS
LIN {X 0.104,Y -261.773,Z 1146.312,A 0.000,B 0.000,C 90.000,E1 56.087} C_DIS
LIN {X -0.111,Y -250.089,Z 1146.292,A 0.000,B 0.000,C 90.000,E1 52.557} C_DIS
LIN {X -0.048,Y -240.395,Z 1146.274,A 0.000,B 0.000,C 90.000,E1 49.256} C_DIS
LIN {X -0.019,Y -230.533,Z 1146.253,A 0.000,B 0.000,C 90.000,E1 45.526} C_DIS
LIN {X -0.130,Y -221.281,Z 1146.232,A 0.000,B 0.000,C 90.000,E1 41.757} C_DIS
LIN {X -0.008,Y -212.647,Z 1146.210,A 0.000,B 0.000,C 90.000,E1 37.855} C_DIS
LIN {X -0.006,Y -204.672,Z 1146.188,A 0.000,B 0.000,C 90.000,E1 33.913} C_DIS
LIN {X -0.072,Y -197.479,Z 1146.166,A 0.000,B 0.000,C 90.000,E1 29.922} C_DIS
LIN {X -0.063,Y -192.386,Z 1146.148,A 0.000,B 0.000,C 90.000,E1 26.668} C_DIS
LIN {X -0.089,Y -187.905,Z 1146.130,A 0.000,B 0.000,C 90.000,E1 23.387} C_DIS
LIN {X -0.039,Y -183.136,Z 1146.107,A 0.000,B 0.000,C 90.000,E1 19.214} C_DIS
LIN {X -0.025,Y -179.310,Z 1146.083,A 0.000,B 0.000,C 90.000,E1 15.009} C_DIS
LIN {X 0.030,Y -176.157,Z 1146.055,A 0.000,B 0.000,C 90.000,E1 9.905} C_DIS
LIN {X -0.022,Y -174.196,Z 1146.012,A 0.000,B 0.000,C 90.000,E1 2.236} C_DIS
LIN {X -0.084,Y -175.923,Z 1145.964,A 0.000,B 0.000,C 90.000,E1 353.571} C_DIS
LIN {X -0.092,Y -178.950,Z 1145.936,A 0.000,B 0.000,C 90.000,E1 348.465} C_DIS
LIN {X -0.011,Y -182.487,Z 1145.912,A 0.000,B 0.000,C 90.000,E1 344.212} C_DIS
LIN {X 0.033,Y -186.925,Z 1145.889,A 0.000,B 0.000,C 90.000,E1 340.007} C_DIS
LIN {X 0.003,Y -192.152,Z 1145.866,A 0.000,B 0.000,C 90.000,E1 335.869} C_DIS
LIN {X 0.010,Y -198.206,Z 1145.843,A 0.000,B 0.000,C 90.000,E1 331.769} C_DIS
LIN {X -0.003,Y -203.692,Z 1145.825,A 0.000,B 0.000,C 90.000,E1 328.535} C_DIS
LIN {X 0.097,Y -209.801,Z 1145.807,A 0.000,B 0.000,C 90.000,E1 325.308} C_DIS
LIN {X -0.042,Y -216.703,Z 1145.790,A 0.000,B 0.000,C 90.000,E1 322.190} C_DIS
LIN {X -0.095,Y -224.508,Z 1145.773,A 0.000,B 0.000,C 90.000,E1 319.094} C_DIS
LIN {X -0.140,Y -233.274,Z 1145.756,A 0.000,B 0.000,C 90.000,E1 316.053} C_DIS
LIN {X 0.044,Y -243.006,Z 1145.739,A 0.000,B 0.000,C 90.000,E1 313.014} C_DIS
LIN {X -0.010,Y -253.914,Z 1145.723,A 0.000,B 0.000,C 90.000,E1 310.092} C_DIS
LIN {X -0.082,Y -266.038,Z 1145.707,A 0.000,B 0.000,C 90.000,E1 307.237} C_DIS
LIN {X 0.004,Y -281.337,Z 1145.689,A 0.000,B 0.000,C 90.000,E1 304.072} C_DIS
LIN {X 0.101,Y -292.525,Z 1145.678,A 0.000,B 0.000,C 90.000,E1 302.005} C_DIS
LIN {X 0.151,Y -308.577,Z 1145.663,A 0.000,B 0.000,C 90.000,E1 299.333} C_DIS
LIN {X 0.171,Y -326.362,Z 1145.649,A 0.000,B 0.000,C 90.000,E1 296.744} C_DIS
LIN {X -0.029,Y -341.093,Z 1145.638,A 0.000,B 0.000,C 90.000,E1 294.899} C_DIS
LIN {X 0.198,Y -353.773,Z 1145.630,A 0.000,B 0.000,C 90.000,E1 293.387} C_DIS
LIN {X 0.092,Y -367.066,Z 1145.622,A 0.000,B 0.000,C 90.000,E1 292.025} C_DIS
LIN {X 0.067,Y -391.578,Z 1145.610,A 0.000,B 0.000,C 90.000,E1 289.758} C_DIS
LIN {X 0.082,Y -402.323,Z 1145.604,A 0.000,B 0.000,C 90.000,E1 288.779} C_DIS
LIN {X -0.203,Y -412.818,Z 1145.599,A 0.000,B 0.000,C 90.000,E1 287.819} C_DIS
LIN {X -0.144,Y -422.897,Z 1145.593,A 0.000,B 0.000,C 90.000,E1 286.804} C_DIS
LIN {X -0.194,Y -430.369,Z 1145.589,A 0.000,B 0.000,C 90.000,E1 286.024} C_DIS
LIN {X 0.061,Y -437.503,Z 1145.584,A 0.000,B 0.000,C 90.000,E1 285.190} C_DIS
LIN {X -0.075,Y -443.980,Z 1145.580,A 0.000,B 0.000,C 90.000,E1 284.411} C_DIS
LIN {X 0.162,Y -449.834,Z 1145.576,A 0.000,B 0.000,C 90.000,E1 283.592} C_DIS
LIN {X 0.024,Y -454.931,Z 1145.571,A 0.000,B 0.000,C 90.000,E1 282.827} C_DIS
LIN {X -0.076,Y -459.368,Z 1145.567,A 0.000,B 0.000,C 90.000,E1 282.063} C_DIS
LIN {X -0.136,Y -463.211,Z 1145.563,A 0.000,B 0.000,C 90.000,E1 281.299} C_DIS
LIN {X 0.203,Y -466.579,Z 1145.558,A 0.000,B 0.000,C 90.000,E1 280.489} C_DIS
LIN {X -0.107,Y -468.570,Z 1145.556,A 0.000,B 0.000,C 90.000,E1 280.018} C_DIS
LIN {X -0.032,Y -470.379,Z 1145.553,A 0.000,B 0.000,C 90.000,E1 279.500} C_DIS
LIN {X 0.132,Y -471.955,Z 1145.550,A 0.000,B 0.000,C 90.000,E1 278.973} C_DIS
LIN {X -0.234,Y -473.265,Z 1145.547,A 0.000,B 0.000,C 90.000,E1 278.511} C_DIS
LIN {X -0.122,Y -474.291,Z 1145.544,A 0.000,B 0.000,C 90.000,E1 277.992} C_DIS
LIN {X 0.062,Y -475.007,Z 1145.542,A 0.000,B 0.000,C 90.000,E1 277.466} C_DIS
LIN {X 0.189,Y -475.374,Z 1145.539,A 0.000,B 0.000,C 90.000,E1 276.947} C_DIS
LIN {X -0.152,Y -475.378,Z 1145.536,A 0.000,B 0.000,C 90.000,E1 276.486} C_DIS
LIN {X -0.020,Y -474.983,Z 1145.533,A 0.000,B 0.000,C 90.000,E1 275.967} C_DIS
LIN {X 0.068,Y -474.118,Z 1145.530,A 0.000,B 0.000,C 90.000,E1 275.454} C_DIS
LIN {X 0.200,Y -472.901,Z 1145.528,A 0.000,B 0.000,C 90.000,E1 274.935} C_DIS
LIN {X -0.145,Y -471.227,Z 1145.525,A 0.000,B 0.000,C 90.000,E1 274.473} C_DIS
LIN {X -0.030,Y -469.017,Z 1145.522,A 0.000,B 0.000,C 90.000,E1 273.955} C_DIS
LIN {X 0.038,Y -466.123,Z 1145.519,A 0.000,B 0.000,C 90.000,E1 273.440} C_DIS
LIN {X -0.166,Y -464.445,Z 1145.518,A 0.000,B 0.000,C 90.000,E1 273.212} C_DIS
LIN {X -0.093,Y -460.294,Z 1145.515,A 0.000,B 0.000,C 90.000,E1 272.694} C_DIS
LIN {X 0.156,Y -457.851,Z 1145.513,A 0.000,B 0.000,C 90.000,E1 272.407} C_DIS
LIN {X -0.061,Y -455.018,Z 1145.512,A 0.000,B 0.000,C 90.000,E1 272.178} C_DIS
LIN {X 0.178,Y -451.831,Z 1145.511,A 0.000,B 0.000,C 90.000,E1 271.892} C_DIS
LIN {X -0.069,Y -445.325,Z 1145.508,A 0.000,B 0.000,C 90.000,E1 271.489} C_DIS
LIN {X -0.207,Y -438.454,Z 1145.506,A 0.000,B 0.000,C 90.000,E1 271.146} C_DIS
LIN {X 0.133,Y -431.430,Z 1145.505,A 0.000,B 0.000,C 90.000,E1 270.802} C_DIS
LIN {X -0.005,Y -424.387,Z 1145.503,A 0.000,B 0.000,C 90.000,E1 270.573} C_DIS
LIN {X 0.138,Y -417.149,Z 1145.502,A 0.000,B 0.000,C 90.000,E1 270.344} C_DIS
LIN {X 0.110,Y -409.908,Z 1145.501,A 0.000,B 0.000,C 90.000,E1 270.172} C_DIS
LIN {X -0.174,Y -398.988,Z 1145.500,A 0.000,B 0.000,C 90.000,E1 270.000} C_DIS
LIN {X 0.189,Y -390.905,Z 1145.499,A 0.000,B 0.000,C 90.000,E1 269.828} C_DIS
LIN {X 0.097,Y -380.501,Z 1145.499,A 0.000,B 0.000,C 90.000,E1 269.771} C_DIS
LIN {X -0.007,Y -373.372,Z 1145.499,A 0.000,B 0.000,C 90.000,E1 269.771} C_DIS
LIN {X -0.028,Y -181.508,Z 1145.499,A 0.000,B 0.000,C 90.000,E1 269.771} C_DIS
LIN {X 0.060,Y -180.896,Z 1145.473,A 0.000,B 0.000,C 90.000,E1 265.179} C_DIS
LIN {X 0.067,Y -179.839,Z 1145.459,A 0.000,B 0.000,C 90.000,E1 262.648} C_DIS
LIN {X -0.055,Y -179.025,Z 1145.445,A 0.000,B 0.000,C 90.000,E1 260.151} C_DIS
LIN {X 0.007,Y -178.667,Z 1145.440,A 0.000,B 0.000,C 90.000,E1 259.285} C_DIS
LIN {X -0.056,Y -175.717,Z 1145.412,A 0.000,B 0.000,C 90.000,E1 254.212} C_DIS
LIN {X -0.040,Y -172.433,Z 1145.388,A 0.000,B 0.000,C 90.000,E1 249.934} C_DIS
LIN {X -0.021,Y -171.261,Z 1145.379,A 0.000,B 0.000,C 90.000,E1 248.209} C_DIS
LIN {X -0.037,Y -167.533,Z 1145.355,A 0.000,B 0.000,C 90.000,E1 243.896} C_DIS
LIN {X 0.045,Y -166.927,Z 1145.350,A 0.000,B 0.000,C 90.000,E1 242.999} C_DIS
LIN {X -0.033,Y -162.924,Z 1145.326,A 0.000,B 0.000,C 90.000,E1 238.663} C_DIS
LIN {X -0.055,Y -161.597,Z 1145.316,A 0.000,B 0.000,C 90.000,E1 236.914} C_DIS
LIN {X 0.070,Y -158.340,Z 1145.297,A 0.000,B 0.000,C 90.000,E1 233.336} C_DIS
LIN {X -0.068,Y -155.642,Z 1145.277,A 0.000,B 0.000,C 90.000,E1 229.828} C_DIS
LIN {X -0.015,Y -151.914,Z 1145.252,A 0.000,B 0.000,C 90.000,E1 225.324} C_DIS
LIN {X 0.000,Y -150.148,Z 1145.237,A 0.000,B 0.000,C 90.000,E1 222.609} C_DIS
LIN {X -0.079,Y -146.931,Z 1145.211,A 0.000,B 0.000,C 90.000,E1 218.096} C_DIS
LIN {X 0.028,Y -145.519,Z 1145.196,A 0.000,B 0.000,C 90.000,E1 215.311} C_DIS
LIN {X 0.023,Y -142.920,Z 1145.171,A 0.000,B 0.000,C 90.000,E1 210.718} C_DIS
LIN {X 0.075,Y -141.542,Z 1145.150,A 0.000,B 0.000,C 90.000,E1 207.001} C_DIS
LIN {X -0.061,Y -139.402,Z 1145.114,A 0.000,B 0.000,C 90.000,E1 200.556} C_DIS
LIN {X -0.008,Y -139.119,Z 1145.104,A 0.000,B 0.000,C 90.000,E1 198.671} C_DIS
LIN {X 0.024,Y -138.352,Z 1145.057,A 0.000,B 0.000,C 90.000,E1 190.254} C_DIS
LIN {X 0.014,Y -139.504,Z 1145.005,A 0.000,B 0.000,C 90.000,E1 180.917} C_DIS
LIN {X -0.045,Y -141.136,Z 1144.974,A 0.000,B 0.000,C 90.000,E1 175.355} C_DIS
LIN {X 0.049,Y -142.516,Z 1144.959,A 0.000,B 0.000,C 90.000,E1 172.534} C_DIS
LIN {X -0.005,Y -144.778,Z 1144.933,A 0.000,B 0.000,C 90.000,E1 167.937} C_DIS
LIN {X -0.057,Y -147.392,Z 1144.913,A 0.000,B 0.000,C 90.000,E1 164.283} C_DIS
LIN {X 0.005,Y -150.723,Z 1144.887,A 0.000,B 0.000,C 90.000,E1 159.699} C_DIS
LIN {X -0.055,Y -154.204,Z 1144.867,A 0.000,B 0.000,C 90.000,E1 156.102} C_DIS
LIN {X 0.014,Y -157.644,Z 1144.847,A 0.000,B 0.000,C 90.000,E1 152.487} C_DIS
LIN {X -0.038,Y -161.904,Z 1144.827,A 0.000,B 0.000,C 90.000,E1 148.948} C_DIS
LIN {X 0.070,Y -166.095,Z 1144.808,A 0.000,B 0.000,C 90.000,E1 145.388} C_DIS
LIN {X 0.067,Y -171.104,Z 1144.788,A 0.000,B 0.000,C 90.000,E1 141.904} C_DIS
LIN {X -0.013,Y -175.979,Z 1144.769,A 0.000,B 0.000,C 90.000,E1 138.485} C_DIS
LIN {X 0.101,Y -180.224,Z 1144.755,A 0.000,B 0.000,C 90.000,E1 135.891} C_DIS
LIN {X 0.076,Y -185.639,Z 1144.736,A 0.000,B 0.000,C 90.000,E1 132.528} C_DIS
LIN {X 0.007,Y -190.236,Z 1144.723,A 0.000,B 0.000,C 90.000,E1 130.048} C_DIS
LIN {X 0.020,Y -197.565,Z 1144.700,A 0.000,B 0.000,C 90.000,E1 125.931} C_DIS
LIN {X -0.099,Y -201.204,Z 1144.689,A 0.000,B 0.000,C 90.000,E1 124.119} C_DIS
LIN {X 0.056,Y -310.904,Z 1144.689,A 0.000,B 0.000,C 90.000,E1 124.072} C_DIS
LIN {X -0.090,Y -312.362,Z 1144.689,A 0.000,B 0.000,C 90.000,E1 124.072} C_DIS
LIN {X -0.041,Y -317.774,Z 1144.688,A 0.000,B 0.000,C 90.000,E1 123.785} C_DIS
LIN {X 0.008,Y -320.627,Z 1144.686,A 0.000,B 0.000,C 90.000,E1 123.499} C_DIS
LIN {X -0.027,Y -324.278,Z 1144.683,A 0.000,B 0.000,C 90.000,E1 122.959} C_DIS
LIN {X 0.058,Y -325.756,Z 1144.681,A 0.000,B 0.000,C 90.000,E1 122.625} C_DIS
LIN {X 0.012,Y -337.789,Z 1144.664,A 0.000,B 0.000,C 90.000,E1 119.489} C_DIS
LIN {X -0.158,Y -350.021,Z 1144.648,A 0.000,B 0.000,C 90.000,E1 116.744} C_DIS
LIN {X 0.007,Y -363.734,Z 1144.633,A 0.000,B 0.000,C 90.000,E1 114.003} C_DIS
LIN {X -0.131,Y -377.269,Z 1144.620,A 0.000,B 0.000,C 90.000,E1 111.663} C_DIS
LIN {X 0.075,Y -392.167,Z 1144.607,A 0.000,B 0.000,C 90.000,E1 109.322} C_DIS
LIN {X -0.116,Y -408.535,Z 1144.595,A 0.000,B 0.000,C 90.000,E1 107.094} C_DIS
LIN {X -0.141,Y -426.488,Z 1144.583,A 0.000,B 0.000,C 90.000,E1 104.898} C_DIS
LIN {X -0.134,Y -446.011,Z 1144.571,A 0.000,B 0.000,C 90.000,E1 102.771} C_DIS
LIN {X 0.055,Y -466.277,Z 1144.560,A 0.000,B 0.000,C 90.000,E1 100.782} C_DIS
LIN {X 0.061,Y -468.846,Z 1144.559,A 0.000,B 0.000,C 90.000,E1 100.546} C_DIS
LIN {X 0.069,Y -470.945,Z 1144.557,A 0.000,B 0.000,C 90.000,E1 100.310} C_DIS
LIN {X 0.076,Y -472.537,Z 1144.556,A 0.000,B 0.000,C 90.000,E1 100.074} C_DIS
LIN {X -0.147,Y -473.839,Z 1144.555,A 0.000,B 0.000,C 90.000,E1 99.849} C_DIS
LIN {X 0.177,Y -474.799,Z 1144.553,A 0.000,B 0.000,C 90.000,E1 99.557} C_DIS
LIN {X -0.170,Y -475.870,Z 1144.550,A 0.000,B 0.000,C 90.000,E1 99.095} C_DIS
LIN {X 0.030,Y -475.949,Z 1144.548,A 0.000,B 0.000,C 90.000,E1 98.568} C_DIS
LIN {X 0.165,Y -475.053,Z 1144.545,A 0.000,B 0.000,C 90.000,E1 98.049} C_DIS
LIN {X -0.167,Y -473.033,Z 1144.542,A 0.000,B 0.000,C 90.000,E1 97.587} C_DIS
LIN {X 0.163,Y -471.475,Z 1144.541,A 0.000,B 0.000,C 90.000,E1 97.296} C_DIS
LIN {X -0.175,Y -455.110,Z 1144.528,A 0.000,B 0.000,C 90.000,E1 95.049} C_DIS
LIN {X 0.117,Y -437.810,Z 1144.513,A 0.000,B 0.000,C 90.000,E1 92.407} C_DIS
LIN {X 0.109,Y -418.699,Z 1144.496,A 0.000,B 0.000,C 90.000,E1 89.198} C_DIS
LIN {X -0.053,Y -408.475,Z 1144.485,A 0.000,B 0.000,C 90.000,E1 87.306} C_DIS
LIN {X -0.040,Y -399.479,Z 1144.476,A 0.000,B 0.000,C 90.000,E1 85.641} C_DIS
LIN {X -0.088,Y -386.072,Z 1144.462,A 0.000,B 0.000,C 90.000,E1 83.109} C_DIS
LIN {X -0.012,Y -377.154,Z 1144.452,A 0.000,B 0.000,C 90.000,E1 81.376} C_DIS
LIN {X -0.041,Y -367.940,Z 1144.442,A 0.000,B 0.000,C 90.000,E1 79.634} C_DIS
LIN {X -0.168,Y -358.389,Z 1144.432,A 0.000,B 0.000,C 90.000,E1 77.881} C_DIS
LIN {X -0.030,Y -346.895,Z 1144.421,A 0.000,B 0.000,C 90.000,E1 75.755} C_DIS
LIN {X -0.042,Y -335.449,Z 1144.409,A 0.000,B 0.000,C 90.000,E1 73.614} C_DIS
LIN {X 0.014,Y -321.202,Z 1144.393,A 0.000,B 0.000,C 90.000,E1 70.786} C_DIS
LIN {X 0.108,Y -304.870,Z 1144.374,A 0.000,B 0.000,C 90.000,E1 67.230} C_DIS
LIN {X 0.128,Y -293.695,Z 1144.359,A 0.000,B 0.000,C 90.000,E1 64.588} C_DIS
LIN {X 0.091,Y -281.532,Z 1144.342,A 0.000,B 0.000,C 90.000,E1 61.563} C_DIS
LIN {X 0.126,Y -269.966,Z 1144.325,A 0.000,B 0.000,C 90.000,E1 58.456} C_DIS
LIN {X -0.016,Y -260.150,Z 1144.309,A 0.000,B 0.000,C 90.000,E1 55.674} C_DIS
LIN {X 0.071,Y -248.558,Z 1144.289,A 0.000,B 0.000,C 90.000,E1 52.065} C_DIS
LIN {X 0.042,Y -237.952,Z 1144.269,A 0.000,B 0.000,C 90.000,E1 48.405} C_DIS
LIN {X -0.009,Y -228.239,Z 1144.248,A 0.000,B 0.000,C 90.000,E1 44.676} C_DIS
LIN {X -0.018,Y -219.109,Z 1144.227,A 0.000,B 0.000,C 90.000,E1 40.862} C_DIS
LIN {X 0.069,Y -210.574,Z 1144.205,A 0.000,B 0.000,C 90.000,E1 36.950} C_DIS
LIN {X 0.076,Y -204.227,Z 1144.188,A 0.000,B 0.000,C 90.000,E1 33.785} C_DIS
LIN {X -0.003,Y -197.033,Z 1144.166,A 0.000,B 0.000,C 90.000,E1 29.795} C_DIS
LIN {X -0.005,Y -191.957,Z 1144.147,A 0.000,B 0.000,C 90.000,E1 26.539} C_DIS
LIN {X 0.028,Y -186.461,Z 1144.125,A 0.000,B 0.000,C 90.000,E1 22.408} C_DIS
LIN {X 0.033,Y -181.903,Z 1144.101,A 0.000,B 0.000,C 90.000,E1 18.236} C_DIS
LIN {X 0.078,Y -178.310,Z 1144.078,A 0.000,B 0.000,C 90.000,E1 14.008} C_DIS
LIN {X 0.062,Y -175.421,Z 1144.050,A 0.000,B 0.000,C 90.000,E1 8.916} C_DIS
LIN {X 0.077,Y -175.611,Z 1143.964,A 0.000,B 0.000,C 90.000,E1 353.514} C_DIS
LIN {X 0.058,Y -178.611,Z 1143.936,A 0.000,B 0.000,C 90.000,E1 348.409} C_DIS
LIN {X -0.048,Y -182.139,Z 1143.912,A 0.000,B 0.000,C 90.000,E1 344.212} C_DIS
LIN {X -0.015,Y -186.579,Z 1143.889,A 0.000,B 0.000,C 90.000,E1 340.007} C_DIS
LIN {X 0.021,Y -191.774,Z 1143.866,A 0.000,B 0.000,C 90.000,E1 335.845} C_DIS
LIN {X -0.064,Y -197.859,Z 1143.843,A 0.000,B 0.000,C 90.000,E1 331.769} C_DIS
LIN {X -0.089,Y -203.352,Z 1143.825,A 0.000,B 0.000,C 90.000,E1 328.535} C_DIS
LIN {X 0.002,Y -209.491,Z 1143.807,A 0.000,B 0.000,C 90.000,E1 325.308} C_DIS
LIN {X 0.022,Y -216.472,Z 1143.790,A 0.000,B 0.000,C 90.000,E1 322.145} C_DIS
LIN {X 0.104,Y -224.275,Z 1143.772,A 0.000,B 0.000,C 90.000,E1 319.013} C_DIS
LIN {X 0.063,Y -233.059,Z 1143.755,A 0.000,B 0.000,C 90.000,E1 315.972} C_DIS
LIN {X -0.094,Y -242.839,Z 1143.739,A 0.000,B 0.000,C 90.000,E1 313.014} C_DIS
LIN {X -0.158,Y -253.785,Z 1143.723,A 0.000,B 0.000,C 90.000,E1 310.092} C_DIS
LIN {X 0.133,Y -266.002,Z 1143.707,A 0.000,B 0.000,C 90.000,E1 307.156} C_DIS
LIN {X -0.007,Y -281.374,Z 1143.689,A 0.000,B 0.000,C 90.000,E1 304.040} C_DIS
LIN {X -0.073,Y -292.578,Z 1143.678,A 0.000,B 0.000,C 90.000,E1 302.005} C_DIS
LIN {X -0.029,Y -308.684,Z 1143.663,A 0.000,B 0.000,C 90.000,E1 299.333} C_DIS
LIN {X -0.018,Y -326.508,Z 1143.649,A 0.000,B 0.000,C 90.000,E1 296.744} C_DIS
LIN {X 0.082,Y -341.246,Z 1143.638,A 0.000,B 0.000,C 90.000,E1 294.847} C_DIS
LIN {X -0.023,Y -353.976,Z 1143.630,A 0.000,B 0.000,C 90.000,E1 293.387} C_DIS
LIN {X -0.108,Y -367.267,Z 1143.622,A 0.000,B 0.000,C 90.000,E1 292.025} C_DIS
LIN {X -0.097,Y -391.708,Z 1143.610,A 0.000,B 0.000,C 90.000,E1 289.758} C_DIS
LIN {X -0.044,Y -402.407,Z 1143.604,A 0.000,B 0.000,C 90.000,E1 288.779} C_DIS
LIN {X 0.164,Y -412.779,Z 1143.599,A 0.000,B 0.000,C 90.000,E1 287.764} C_DIS
LIN {X 0.221,Y -423.054,Z 1143.593,A 0.000,B 0.000,C 90.000,E1 286.732} C_DIS
LIN {X 0.087,Y -430.481,Z 1143.589,A 0.000,B 0.000,C 90.000,E1 285.969} C_DIS
LIN {X -0.059,Y -437.597,Z 1143.584,A 0.000,B 0.000,C 90.000,E1 285.190} C_DIS
LIN {X 0.235,Y -444.126,Z 1143.580,A 0.000,B 0.000,C 90.000,E1 284.356} C_DIS
LIN {X 0.041,Y -449.999,Z 1143.576,A 0.000,B 0.000,C 90.000,E1 283.592} C_DIS
LIN {X -0.096,Y -455.096,Z 1143.571,A 0.000,B 0.000,C 90.000,E1 282.827} C_DIS
LIN {X -0.197,Y -459.552,Z 1143.567,A 0.000,B 0.000,C 90.000,E1 282.063} C_DIS
LIN {X 0.199,Y -463.443,Z 1143.563,A 0.000,B 0.000,C 90.000,E1 281.243} C_DIS
LIN {X 0.085,Y -466.806,Z 1143.558,A 0.000,B 0.000,C 90.000,E1 280.489} C_DIS
LIN {X -0.150,Y -470.632,Z 1143.553,A 0.000,B 0.000,C 90.000,E1 279.500} C_DIS
LIN {X 0.017,Y -472.213,Z 1143.550,A 0.000,B 0.000,C 90.000,E1 278.973} C_DIS
LIN {X 0.120,Y -473.503,Z 1143.547,A 0.000,B 0.000,C 90.000,E1 278.454} C_DIS
LIN {X -0.235,Y -474.523,Z 1143.544,A 0.000,B 0.000,C 90.000,E1 277.992} C_DIS
LIN {X -0.050,Y -475.230,Z 1143.542,A 0.000,B 0.000,C 90.000,E1 277.466} C_DIS
LIN {X 0.078,Y -475.612,Z 1143.539,A 0.000,B 0.000,C 90.000,E1 276.947} C_DIS
LIN {X 0.211,Y -475.564,Z 1143.536,A 0.000,B 0.000,C 90.000,E1 276.429} C_DIS
LIN {X -0.128,Y -475.202,Z 1143.533,A 0.000,B 0.000,C 90.000,E1 275.967} C_DIS
LIN {X -0.040,Y -474.348,Z 1143.530,A 0.000,B 0.000,C 90.000,E1 275.454} C_DIS
LIN {X 0.095,Y -473.184,Z 1143.527,A 0.000,B 0.000,C 90.000,E1 274.935} C_DIS
LIN {X 0.220,Y -471.509,Z 1143.525,A 0.000,B 0.000,C 90.000,E1 274.416} C_DIS
LIN {X -0.131,Y -469.282,Z 1143.522,A 0.000,B 0.000,C 90.000,E1 273.955} C_DIS
LIN {X 0.136,Y -468.009,Z 1143.521,A 0.000,B 0.000,C 90.000,E1 273.669} C_DIS
LIN {X 0.200,Y -464.818,Z 1143.518,A 0.000,B 0.000,C 90.000,E1 273.154} C_DIS
LIN {X -0.188,Y -460.703,Z 1143.515,A 0.000,B 0.000,C 90.000,E1 272.694} C_DIS
LIN {X 0.063,Y -458.291,Z 1143.513,A 0.000,B 0.000,C 90.000,E1 272.407} C_DIS
LIN {X -0.156,Y -455.461,Z 1143.512,A 0.000,B 0.000,C 90.000,E1 272.178} C_DIS
LIN {X 0.081,Y -452.265,Z 1143.511,A 0.000,B 0.000,C 90.000,E1 271.892} C_DIS
LIN {X -0.159,Y -445.823,Z 1143.508,A 0.000,B 0.000,C 90.000,E1 271.489} C_DIS
LIN {X 0.126,Y -438.959,Z 1143.506,A 0.000,B 0.000,C 90.000,E1 271.088} C_DIS
LIN {X 0.003,Y -431.899,Z 1143.505,A 0.000,B 0.000,C 90.000,E1 270.802} C_DIS
LIN {X -0.155,Y -424.815,Z 1143.503,A 0.000,B 0.000,C 90.000,E1 270.573} C_DIS
LIN {X -0.009,Y -417.690,Z 1143.502,A 0.000,B 0.000,C 90.000,E1 270.344} C_DIS
LIN {X -0.167,Y -406.735,Z 1143.500,A 0.000,B 0.000,C 90.000,E1 270.115} C_DIS
LIN {X 0.046,Y -395.487,Z 1143.499,A 0.000,B 0.000,C 90.000,E1 269.885} C_DIS
LIN {X -0.119,Y -388.395,Z 1143.499,A 0.000,B 0.000,C 90.000,E1 269.828} C_DIS
LIN {X -0.077,Y -377.630,Z 1143.499,A 0.000,B 0.000,C 90.000,E1 269.771} C_DIS
LIN {X -0.129,Y -372.303,Z 1143.499,A 0.000,B 0.000,C 90.000,E1 269.771} C_DIS
LIN {X -0.088,Y -181.503,Z 1143.499,A 0.000,B 0.000,C 90.000,E1 269.771} C_DIS
LIN {X -0.003,Y -180.893,Z 1143.473,A 0.000,B 0.000,C 90.000,E1 265.179} C_DIS
LIN {X 0.075,Y -179.517,Z 1143.454,A 0.000,B 0.000,C 90.000,E1 261.781} C_DIS
LIN {X 0.059,Y -179.020,Z 1143.445,A 0.000,B 0.000,C 90.000,E1 260.095} C_DIS
LIN {X -0.055,Y -178.654,Z 1143.440,A 0.000,B 0.000,C 90.000,E1 259.285} C_DIS
LIN {X 0.051,Y -175.705,Z 1143.412,A 0.000,B 0.000,C 90.000,E1 254.157} C_DIS
LIN {X 0.062,Y -172.420,Z 1143.388,A 0.000,B 0.000,C 90.000,E1 249.880} C_DIS
LIN {X 0.077,Y -171.241,Z 1143.379,A 0.000,B 0.000,C 90.000,E1 248.156} C_DIS
LIN {X 0.053,Y -167.518,Z 1143.355,A 0.000,B 0.000,C 90.000,E1 243.845} C_DIS
LIN {X -0.015,Y -166.914,Z 1143.350,A 0.000,B 0.000,C 90.000,E1 242.999} C_DIS
LIN {X 0.038,Y -162.222,Z 1143.321,A 0.000,B 0.000,C 90.000,E1 237.740} C_DIS
LIN {X -0.043,Y -160.803,Z 1143.311,A 0.000,B 0.000,C 90.000,E1 236.008} C_DIS
LIN {X -0.065,Y -157.591,Z 1143.291,A 0.000,B 0.000,C 90.000,E1 232.477} C_DIS
LIN {X -0.007,Y -155.624,Z 1143.277,A 0.000,B 0.000,C 90.000,E1 229.784} C_DIS
LIN {X -0.072,Y -151.900,Z 1143.252,A 0.000,B 0.000,C 90.000,E1 225.324} C_DIS
LIN {X -0.056,Y -150.130,Z 1143.237,A 0.000,B 0.000,C 90.000,E1 222.609} C_DIS
LIN {X 0.072,Y -146.919,Z 1143.211,A 0.000,B 0.000,C 90.000,E1 218.016} C_DIS
LIN {X -0.027,Y -145.507,Z 1143.196,A 0.000,B 0.000,C 90.000,E1 215.311} C_DIS
LIN {X -0.031,Y -142.910,Z 1143.171,A 0.000,B 0.000,C 90.000,E1 210.718} C_DIS
LIN {X 0.021,Y -141.531,Z 1143.150,A 0.000,B 0.000,C 90.000,E1 207.001} C_DIS
LIN {X 0.064,Y -139.399,Z 1143.114,A 0.000,B 0.000,C 90.000,E1 200.482} C_DIS
LIN {X -0.016,Y -139.112,Z 1143.104,A 0.000,B 0.000,C 90.000,E1 198.652} C_DIS
LIN {X -0.029,Y -138.352,Z 1143.057,A 0.000,B 0.000,C 90.000,E1 190.254} C_DIS
LIN {X -0.040,Y -139.507,Z 1143.005,A 0.000,B 0.000,C 90.000,E1 180.917} C_DIS
LIN {X 0.042,Y -141.146,Z 1142.974,A 0.000,B 0.000,C 90.000,E1 175.298} C_DIS
LIN {X -0.006,Y -142.526,Z 1142.958,A 0.000,B 0.000,C 90.000,E1 172.534} C_DIS
LIN {X -0.061,Y -144.791,Z 1142.933,A 0.000,B 0.000,C 90.000,E1 167.937} C_DIS
LIN {X 0.070,Y -147.408,Z 1142.912,A 0.000,B 0.000,C 90.000,E1 164.212} C_DIS
LIN {X -0.043,Y -149.984,Z 1142.892,A 0.000,B 0.000,C 90.000,E1 160.604} C_DIS
LIN {X -0.033,Y -153.309,Z 1142.872,A 0.000,B 0.000,C 90.000,E1 156.975} C_DIS
LIN {X 0.019,Y -155.011,Z 1142.862,A 0.000,B 0.000,C 90.000,E1 155.153} C_DIS
LIN {X 0.042,Y -158.654,Z 1142.842,A 0.000,B 0.000,C 90.000,E1 151.563} C_DIS
LIN {X -0.014,Y -161.932,Z 1142.827,A 0.000,B 0.000,C 90.000,E1 148.918} C_DIS
LIN {X 0.010,Y -166.122,Z 1142.808,A 0.000,B 0.000,C 90.000,E1 145.388} C_DIS
LIN {X 0.007,Y -171.133,Z 1142.788,A 0.000,B 0.000,C 90.000,E1 141.904} C_DIS
LIN {X -0.075,Y -176.009,Z 1142.769,A 0.000,B 0.000,C 90.000,E1 138.485} C_DIS
LIN {X 0.038,Y -180.260,Z 1142.755,A 0.000,B 0.000,C 90.000,E1 135.891} C_DIS
LIN {X 0.011,Y -185.673,Z 1142.736,A 0.000,B 0.000,C 90.000,E1 132.528} C_DIS
LIN {X 0.064,Y -190.274,Z 1142.722,A 0.000,B 0.000,C 90.000,E1 130.011} C_DIS
LIN {X -0.046,Y -197.602,Z 1142.700,A 0.000,B 0.000,C 90.000,E1 125.931} C_DIS
LIN {X -0.096,Y -201.203,Z 1142.689,A 0.000,B 0.000,C 90.000,E1 124.119} C_DIS
LIN {X 0.073,Y -310.710,Z 1142.689,A 0.000,B 0.000,C 90.000,E1 124.072} C_DIS
LIN {X -0.017,Y -313.045,Z 1142.689,A 0.000,B 0.000,C 90.000,E1 124.040} C_DIS
LIN {X -0.147,Y -317.995,Z 1142.688,A 0.000,B 0.000,C 90.000,E1 123.785} C_DIS
LIN {X -0.098,Y -320.772,Z 1142.686,A 0.000,B 0.000,C 90.000,E1 123.499} C_DIS
LIN {X -0.201,Y -324.415,Z 1142.683,A 0.000,B 0.000,C 90.000,E1 122.959} C_DIS
LIN {X -0.116,Y -325.858,Z 1142.681,A 0.000,B 0.000,C 90.000,E1 122.625} C_DIS
LIN {X 0.001,Y -337.891,Z 1142.664,A 0.000,B 0.000,C 90.000,E1 119.461} C_DIS
LIN {X -0.026,Y -350.137,Z 1142.648,A 0.000,B 0.000,C 90.000,E1 116.693} C_DIS
LIN {X 0.155,Y -363.867,Z 1142.633,A 0.000,B 0.000,C 90.000,E1 113.951} C_DIS
LIN {X 0.172,Y -377.418,Z 1142.620,A 0.000,B 0.000,C 90.000,E1 111.589} C_DIS
LIN {X -0.116,Y -392.333,Z 1142.607,A 0.000,B 0.000,C 90.000,E1 109.322} C_DIS
LIN {X 0.080,Y -408.719,Z 1142.595,A 0.000,B 0.000,C 90.000,E1 107.040} C_DIS
LIN {X 0.182,Y -426.691,Z 1142.583,A 0.000,B 0.000,C 90.000,E1 104.828} C_DIS
LIN {X 0.103,Y -446.232,Z 1142.571,A 0.000,B 0.000,C 90.000,E1 102.715} C_DIS
LIN {X -0.130,Y -469.052,Z 1142.558,A 0.000,B 0.000,C 90.000,E1 100.546} C_DIS
LIN {X -0.131,Y -471.094,Z 1142.557,A 0.000,B 0.000,C 90.000,E1 100.310} C_DIS
LIN {X -0.134,Y -472.644,Z 1142.556,A 0.000,B 0.000,C 90.000,E1 100.074} C_DIS
LIN {X 0.110,Y -473.905,Z 1142.554,A 0.000,B 0.000,C 90.000,E1 99.792} C_DIS
LIN {X -0.033,Y -474.830,Z 1142.553,A 0.000,B 0.000,C 90.000,E1 99.557} C_DIS
LIN {X 0.164,Y -475.844,Z 1142.550,A 0.000,B 0.000,C 90.000,E1 99.029} C_DIS
LIN {X -0.179,Y -475.872,Z 1142.547,A 0.000,B 0.000,C 90.000,E1 98.568} C_DIS
LIN {X -0.044,Y -474.920,Z 1142.545,A 0.000,B 0.000,C 90.000,E1 98.049} C_DIS
LIN {X 0.092,Y -472.832,Z 1142.542,A 0.000,B 0.000,C 90.000,E1 97.530} C_DIS
LIN {X -0.046,Y -471.224,Z 1142.541,A 0.000,B 0.000,C 90.000,E1 97.296} C_DIS
LIN {X 0.071,Y -454.863,Z 1142.528,A 0.000,B 0.000,C 90.000,E1 94.992} C_DIS
LIN {X -0.090,Y -437.565,Z 1142.513,A 0.000,B 0.000,C 90.000,E1 92.407} C_DIS
LIN {X 0.207,Y -419.959,Z 1142.497,A 0.000,B 0.000,C 90.000,E1 89.427} C_DIS
LIN {X 0.150,Y -408.244,Z 1142.485,A 0.000,B 0.000,C 90.000,E1 87.249} C_DIS
LIN {X 0.153,Y -399.248,Z 1142.476,A 0.000,B 0.000,C 90.000,E1 85.584} C_DIS
LIN {X 0.090,Y -385.842,Z 1142.461,A 0.000,B 0.000,C 90.000,E1 83.053} C_DIS
LIN {X 0.157,Y -376.899,Z 1142.452,A 0.000,B 0.000,C 90.000,E1 81.319} C_DIS
LIN {X 0.118,Y -367.676,Z 1142.442,A 0.000,B 0.000,C 90.000,E1 79.577} C_DIS
LIN {X 0.012,Y -359.748,Z 1142.434,A 0.000,B 0.000,C 90.000,E1 78.117} C_DIS
LIN {X 0.176,Y -348.256,Z 1142.422,A 0.000,B 0.000,C 90.000,E1 75.992} C_DIS
LIN {X 0.079,Y -335.153,Z 1142.409,A 0.000,B 0.000,C 90.000,E1 73.559} C_DIS
LIN {X 0.117,Y -320.918,Z 1142.393,A 0.000,B 0.000,C 90.000,E1 70.732} C_DIS
LIN {X -0.092,Y -304.607,Z 1142.373,A 0.000,B 0.000,C 90.000,E1 67.230} C_DIS
LIN {X -0.071,Y -293.430,Z 1142.359,A 0.000,B 0.000,C 90.000,E1 64.588} C_DIS
LIN {X 0.140,Y -281.268,Z 1142.342,A 0.000,B 0.000,C 90.000,E1 61.513} C_DIS
LIN {X -0.071,Y -269.707,Z 1142.325,A 0.000,B 0.000,C 90.000,E1 58.456} C_DIS
LIN {X 0.150,Y -259.881,Z 1142.309,A 0.000,B 0.000,C 90.000,E1 55.595} C_DIS
LIN {X 0.028,Y -248.271,Z 1142.289,A 0.000,B 0.000,C 90.000,E1 52.029} C_DIS
LIN {X 0.003,Y -237.673,Z 1142.269,A 0.000,B 0.000,C 90.000,E1 48.366} C_DIS
LIN {X -0.106,Y -229.837,Z 1142.252,A 0.000,B 0.000,C 90.000,E1 45.405} C_DIS
LIN {X -0.077,Y -220.554,Z 1142.231,A 0.000,B 0.000,C 90.000,E1 41.595} C_DIS
LIN {X 0.061,Y -213.577,Z 1142.214,A 0.000,B 0.000,C 90.000,E1 38.463} C_DIS
LIN {X 0.096,Y -206.988,Z 1142.196,A 0.000,B 0.000,C 90.000,E1 35.311} C_DIS
LIN {X 0.064,Y -200.935,Z 1142.179,A 0.000,B 0.000,C 90.000,E1 32.133} C_DIS
LIN {X -0.089,Y -195.320,Z 1142.161,A 0.000,B 0.000,C 90.000,E1 28.949} C_DIS
LIN {X 0.029,Y -189.284,Z 1142.138,A 0.000,B 0.000,C 90.000,E1 24.823} C_DIS
LIN {X 0.076,Y -184.147,Z 1142.115,A 0.000,B 0.000,C 90.000,E1 20.663} C_DIS
LIN {X -0.004,Y -180.000,Z 1142.092,A 0.000,B 0.000,C 90.000,E1 16.496} C_DIS
LIN {X 0.068,Y -176.849,Z 1142.068,A 0.000,B 0.000,C 90.000,E1 12.243} C_DIS
LIN {X -0.056,Y -174.175,Z 1142.035,A 0.000,B 0.000,C 90.000,E1 6.315} C_DIS
LIN {X 0.063,Y -175.304,Z 1141.964,A 0.000,B 0.000,C 90.000,E1 353.514} C_DIS
LIN {X 0.032,Y -178.285,Z 1141.936,A 0.000,B 0.000,C 90.000,E1 348.409} C_DIS
LIN {X 0.091,Y -181.789,Z 1141.912,A 0.000,B 0.000,C 90.000,E1 344.157} C_DIS
LIN {X -0.063,Y -186.221,Z 1141.889,A 0.000,B 0.000,C 90.000,E1 340.007} C_DIS
LIN {X -0.040,Y -191.399,Z 1141.866,A 0.000,B 0.000,C 90.000,E1 335.845} C_DIS
LIN {X 0.035,Y -197.509,Z 1141.843,A 0.000,B 0.000,C 90.000,E1 331.719} C_DIS
LIN {X -0.002,Y -203.029,Z 1141.825,A 0.000,B 0.000,C 90.000,E1 328.486} C_DIS
LIN {X 0.077,Y -209.193,Z 1141.807,A 0.000,B 0.000,C 90.000,E1 325.261} C_DIS
LIN {X 0.047,Y -216.215,Z 1141.790,A 0.000,B 0.000,C 90.000,E1 322.110} C_DIS
LIN {X 0.065,Y -225.089,Z 1141.770,A 0.000,B 0.000,C 90.000,E1 318.609} C_DIS
LIN {X 0.048,Y -234.011,Z 1141.753,A 0.000,B 0.000,C 90.000,E1 315.567} C_DIS
LIN {X -0.085,Y -243.977,Z 1141.737,A 0.000,B 0.000,C 90.000,E1 312.609} C_DIS
LIN {X 0.073,Y -255.131,Z 1141.720,A 0.000,B 0.000,C 90.000,E1 309.644} C_DIS
LIN {X 0.035,Y -267.609,Z 1141.704,A 0.000,B 0.000,C 90.000,E1 306.790} C_DIS
LIN {X 0.006,Y -283.202,Z 1141.687,A 0.000,B 0.000,C 90.000,E1 303.658} C_DIS
LIN {X 0.132,Y -300.537,Z 1141.670,A 0.000,B 0.000,C 90.000,E1 300.590} C_DIS
LIN {X 0.089,Y -310.985,Z 1141.661,A 0.000,B 0.000,C 90.000,E1 298.949} C_DIS
LIN {X 0.085,Y -326.654,Z 1141.648,A 0.000,B 0.000,C 90.000,E1 296.693} C_DIS
LIN {X -0.008,Y -341.438,Z 1141.638,A 0.000,B 0.000,C 90.000,E1 294.823} C_DIS
LIN {X -0.164,Y -354.536,Z 1141.630,A 0.000,B 0.000,C 90.000,E1 293.334} C_DIS
LIN {X 0.212,Y -367.941,Z 1141.622,A 0.000,B 0.000,C 90.000,E1 291.897} C_DIS
LIN {X -0.102,Y -392.394,Z 1141.609,A 0.000,B 0.000,C 90.000,E1 289.685} C_DIS
LIN {X -0.156,Y -403.052,Z 1141.604,A 0.000,B 0.000,C 90.000,E1 288.725} C_DIS
LIN {X 0.095,Y -410.933,Z 1141.600,A 0.000,B 0.000,C 90.000,E1 287.946} C_DIS
LIN {X 0.243,Y -421.160,Z 1141.594,A 0.000,B 0.000,C 90.000,E1 286.913} C_DIS
LIN {X 0.133,Y -428.689,Z 1141.590,A 0.000,B 0.000,C 90.000,E1 286.150} C_DIS
LIN {X -0.015,Y -435.951,Z 1141.585,A 0.000,B 0.000,C 90.000,E1 285.371} C_DIS
LIN {X -0.170,Y -442.695,Z 1141.581,A 0.000,B 0.000,C 90.000,E1 284.592} C_DIS
LIN {X 0.060,Y -448.736,Z 1141.577,A 0.000,B 0.000,C 90.000,E1 283.772} C_DIS
LIN {X -0.092,Y -454.049,Z 1141.572,A 0.000,B 0.000,C 90.000,E1 283.008} C_DIS
LIN {X -0.195,Y -458.707,Z 1141.568,A 0.000,B 0.000,C 90.000,E1 282.243} C_DIS
LIN {X 0.190,Y -462.729,Z 1141.564,A 0.000,B 0.000,C 90.000,E1 281.422} C_DIS
LIN {X 0.162,Y -466.234,Z 1141.559,A 0.000,B 0.000,C 90.000,E1 280.658} C_DIS
LIN {X 0.072,Y -469.298,Z 1141.555,A 0.000,B 0.000,C 90.000,E1 279.905} C_DIS
LIN {X 0.231,Y -471.093,Z 1141.552,A 0.000,B 0.000,C 90.000,E1 279.378} C_DIS
LIN {X -0.142,Y -472.642,Z 1141.549,A 0.000,B 0.000,C 90.000,E1 278.916} C_DIS
LIN {X -0.036,Y -473.894,Z 1141.547,A 0.000,B 0.000,C 90.000,E1 278.398} C_DIS
LIN {X 0.148,Y -474.869,Z 1141.544,A 0.000,B 0.000,C 90.000,E1 277.871} C_DIS
LIN {X -0.200,Y -475.504,Z 1141.541,A 0.000,B 0.000,C 90.000,E1 277.409} C_DIS
LIN {X -0.070,Y -475.823,Z 1141.538,A 0.000,B 0.000,C 90.000,E1 276.891} C_DIS
LIN {X 0.064,Y -475.779,Z 1141.535,A 0.000,B 0.000,C 90.000,E1 276.372} C_DIS
